	{attribute 'TcIecLibraryType'}
	{attribute 'external_name' := 'F_VN_FindContours_GUID_BC617802_F305_490B_4DCA_5F9C28F7E587'}
	(* Search for object contours in a binary image. Returns only external contours. *)
	FUNCTION F_VN_FindContours : HRESULT
	VAR_INPUT
		ipSrcImage	:	ITcVnImage;	(* Source image (modified by the function) *)
		ipContours	:	REFERENCE TO ITcVnContainer;	(* Returns a container which is filled with the found contours (ContainerType_Vector_Vector_TcVnPoint2_DINT; The elements of this container are single contours. Non-zero interface pointers are reused.) *)
		hrPrev	:	HRESULT;	(* HRESULT indicating the result of previous operations (If SUCCEEDED(hrPrev) equals false, no operation is executed.) *)
	END_VAR

END_FUNCTION

// Functions/Image Analysis/Object Detection/F_VN_FindContoursExp

	{attribute 'TcIecLibraryType'}
	{attribute 'external_name' := 'F_VN_FindContoursExp_GUID_CC63BB9E_985F_4B1D_69D1_A104A588DDE9'}
	(* Search for object contours in a binary image. (expert function) *)
	FUNCTION F_VN_FindContoursExp : HRESULT
	VAR_INPUT
		ipSrcImage	:	ITcVnImage;	(* Source image (modified by the function) *)
		ipContours	:	REFERENCE TO ITcVnContainer;	(* Returns a container which is filled with the found contours (ContainerType_Vector_Vector_TcVnPoint2_DINT; The elements of this container are single contours. Non-zero interface pointers are reused.) *)
		eRetrievalMode	:	ETcVnContourRetrievalMode;	(* Specifies which contours are retrieved and how their relationship is encoded *)
		eApproximationMethod	:	ETcVnContourApproximationMethod;	(* Contour encoding *)
		aOffset	:	REFERENCE TO TcVnPoint;	(* Offset by which every contour point is shifted *)
		hrPrev	:	HRESULT;	(* HRESULT indicating the result of previous operations (If SUCCEEDED(hrPrev) equals false, no operation is executed.) *)
	END_VAR

END_FUNCTION

// Functions/Image Analysis/Object Detection/F_VN_HoughCircles

	{attribute 'TcIecLibraryType'}
	{attribute 'external_name' := 'F_VN_HoughCircles_GUID_86F03E73_E7CE_4817_5925_A59C535A1739'}
	(* Search for circles using the Hough transform. *)
	FUNCTION F_VN_HoughCircles : HRESULT
	VAR_INPUT
		ipSrcImage	:	ITcVnImage;	(* Source image (USINT, 1 channel, gray-level) *)
		ipCircles	:	REFERENCE TO ITcVnContainer;	(* Returns a container which is filled with the found circles (ContainerType_Vector_TcVnVector3_REAL; Each container element contains the x coordinate of the circle center [0], the y coordinate of the circle center [1], and the radius [2], respectively. Non-zero interface pointers are reused.) *)
		fInvAccuRatio	:	LREAL;	(* Inverted ratio of the accumulator size in relation to the source image's size (must be > 0. A value of 2 means that the size is halved in both directions.) *)
		fMinDist	:	LREAL;	(* Smallest allowed distance of two circles (must be > 0) *)
		hrPrev	:	HRESULT;	(* HRESULT indicating the result of previous operations (If SUCCEEDED(hrPrev) equals false, no operation is executed.) *)
	END_VAR

END_FUNCTION

// Functions/Image Analysis/Object Detection/F_VN_HoughCirclesExp

	{attribute 'TcIecLibraryType'}
	{attribute 'external_name' := 'F_VN_HoughCirclesExp_GUID_B1DC5CB1_08D8_43F5_4695_748B5DA9490C'}
	(* Search for circles using the Hough transform. (expert function) *)
	FUNCTION F_VN_HoughCirclesExp : HRESULT
	VAR_INPUT
		ipSrcImage	:	ITcVnImage;	(* Source image (USINT, 1 channel, gray-level) *)
		ipCircles	:	REFERENCE TO ITcVnContainer;	(* Returns a container which is filled with the found circles (ContainerType_Vector_TcVnVector3_REAL; Each container element contains the x coordinate of the circle center [0], the y coordinate of the circle center [1], and the radius [2], respectively. Non-zero interface pointers are reused.) *)
		fInvAccuRatio	:	LREAL;	(* Inverted ratio of the accumulator size in relation to the source image's size (must be > 0. A value of 2 means that the size is halved in both directions.) *)
		fMinDist	:	LREAL;	(* Smallest allowed distance of two circles (must be > 0) *)
		eHoughMethod	:	ETcVnHoughMethod;	(* Hough method to use (currently only valid value: GRADIENT) *)
		fParam1	:	LREAL;	(* First method specific parameter (GRADIENT: upper threshold for canny edge detection, which must be > 0) *)
		fParam2	:	LREAL;	(* Second method specific parameter (GRADIENT: accumulator threshold for detecting circle centers, which must be > 0) *)
		nMinRadius	:	UDINT;	(* Minimum circle radius allowed *)
		nMaxRadius	:	UDINT;	(* Maximum circle radius allowed (if 0, the value is internally set to max(image rows, image columns)) *)
		hrPrev	:	HRESULT;	(* HRESULT indicating the result of previous operations (If SUCCEEDED(hrPrev) equals false, no operation is executed.) *)
	END_VAR

END_FUNCTION

// Functions/Image Analysis/Object Detection/F_VN_HoughLines

	{attribute 'TcIecLibraryType'}
	{attribute 'external_name' := 'F_VN_HoughLines_GUID_3641D244_03BD_44CB_43E4_F0ABC9273C89'}
	(* Search for lines using the standard Hough transform. *)
	FUNCTION F_VN_HoughLines : HRESULT
	VAR_INPUT
		ipSrcImage	:	ITcVnImage;	(* Source image (USINT, 1 channel, binary, may be modified by the function) *)
		ipLines	:	REFERENCE TO ITcVnContainer;	(* Returns a container which is filled with the found lines (ContainerType_Vector_TcVnVector2_REAL; Each container element contains the distance from the origin [0] in pixels and the rotation angle [1] in radians, respectively. Non-zero interface pointers are reused.) *)
		fDistRes	:	LREAL;	(* Distance resolution of the accumulator (in pixels, must be > 0) *)
		fAngleRes	:	LREAL;	(* Angle resolution of the accumulator (in radians, must be > 0) *)
		nAccuThreshold	:	UDINT;	(* Accumulator threshold *)
		hrPrev	:	HRESULT;	(* HRESULT indicating the result of previous operations (If SUCCEEDED(hrPrev) equals false, no operation is executed.) *)
	END_VAR

END_FUNCTION

// Functions/Image Analysis/Object Detection/F_VN_HoughLinesExp

	{attribute 'TcIecLibraryType'}
	{attribute 'external_name' := 'F_VN_HoughLinesExp_GUID_1C9FFE0A_9145_4559_5E8F_3269BB3716B9'}
	(* Search for lines using the standard Hough transform. (expert function) *)
	FUNCTION F_VN_HoughLinesExp : HRESULT
	VAR_INPUT
		ipSrcImage	:	ITcVnImage;	(* Source image (USINT, 1 channel, binary, may be modified by the function) *)
		ipLines	:	REFERENCE TO ITcVnContainer;	(* Returns a container which is filled with the found lines (ContainerType_Vector_TcVnVector2_REAL; Each container element contains the distance from the origin [0] in pixels and the rotation angle [1] in radians, respectively. Non-zero interface pointers are reused.) *)
		fDistRes	:	LREAL;	(* Distance resolution of the accumulator (in pixels, must be > 0) *)
		fAngleRes	:	LREAL;	(* Angle resolution of the accumulator (in radians, must be > 0) *)
		nAccuThreshold	:	UDINT;	(* Accumulator threshold *)
		fDistResDiv	:	LREAL;	(* Divisor of the distance resolution for the multi-scale Hough transform (>= 0, must be > 0 if fAngleResDiv is > 0) *)
		fAngleResDiv	:	LREAL;	(* Divisor of the angle resolution for the multi-scale Hough transform (>= 0, must be > 0 if fDistResDiv is > 0) *)
		hrPrev	:	HRESULT;	(* HRESULT indicating the result of previous operations (If SUCCEEDED(hrPrev) equals false, no operation is executed.) *)
	END_VAR

END_FUNCTION

// Functions/Image Analysis/Object Detection/F_VN_MatchImageHuMoments

	{attribute 'TcIecLibraryType'}
	{attribute 'external_name' := 'F_VN_MatchImageHuMoments_GUID_D174E499_AD66_4F1F_5089_AD3F3CD47605'}
	(* Compare two images using the Hu moment invariants. *)
	FUNCTION F_VN_MatchImageHuMoments : HRESULT
	VAR_INPUT
		ipImage1	:	ITcVnImage;	(* First image (1 channel) *)
		ipImage2	:	ITcVnImage;	(* Second image (1 channel) *)
		eComparisonMethod	:	ETcVnContoursMatchComparisonMethod;	(* Method used for comparing the Hu moment invariants of the images *)
		fDissimilarity	:	REFERENCE TO LREAL;	(* Returns the dissimilarity of the image Hu moment invariants depending on the chosen comparison method *)
		hrPrev	:	HRESULT;	(* HRESULT indicating the result of previous operations (If SUCCEEDED(hrPrev) equals false, no operation is executed.) *)
	END_VAR

END_FUNCTION

// Functions/Image Analysis/Object Detection/F_VN_MatchTemplate

	{attribute 'TcIecLibraryType'}
	{attribute 'external_name' := 'F_VN_MatchTemplate_GUID_741B3C57_0C32_4A22_515B_0F16608AEB4A'}
	(* Match a template image with every location in the source image (using the TCVN_TMM_CCORR_NORMED method) and save the comparison results. *)
	FUNCTION F_VN_MatchTemplate : HRESULT
	VAR_INPUT
		ipSrcImage	:	ITcVnImage;	(* Source image (USINT or REAL, 1 or 3 channels) *)
		ipTemplateImage	:	ITcVnImage;	(* Template image (same type as ipSrcImage, smaller width and height) *)
		ipResultImage	:	REFERENCE TO ITcVnImage;	(* Returns the result image (REAL, normalized to [0..1], 1 channel, dimensions: (ipSrcImage.width - ipTemplateImage.width + 1) x (ipSrcImage.height - ipTemplateImage.height + 1). The best match is the global maximum. The position in ipResultImage is the top-left corner of ipTemplateImage position in ipSrcImage) *)
		hrPrev	:	HRESULT;	(* HRESULT indicating the result of previous operations (If SUCCEEDED(hrPrev) equals false, no operation is executed.) *)
	END_VAR

END_FUNCTION

// Functions/Image Analysis/Object Detection/F_VN_MatchTemplateExp

	{attribute 'TcIecLibraryType'}
	{attribute 'external_name' := 'F_VN_MatchTemplateExp_GUID_82700BC1_22E7_489F_6AAC_8EFF22E27EF5'}
	(* Match a template image with every location in the source image and save the comparison results. (expert function) *)
	FUNCTION F_VN_MatchTemplateExp : HRESULT
	VAR_INPUT
		ipSrcImage	:	ITcVnImage;	(* Source image (USINT or REAL, 1 or 3 channels) *)
		ipTemplateImage	:	ITcVnImage;	(* Template image (same type as ipSrcImage, smaller width and height) *)
		ipResultImage	:	REFERENCE TO ITcVnImage;	(* Returns the result image (REAL, 1 channel, dimensions: (ipSrcImage.width - ipTemplateImage.width + 1) x (ipSrcImage.height - ipTemplateImage.height + 1). The best match is the global minimum (SQDIFF(_NORMED)) or maximum (CCORR(_NORMED), CCOEFF(_NORMED)). The position in ipResultImage is the top-left corner of ipTemplateImage position in ipSrcImage) *)
		eMatchMethod	:	ETcVnTemplateMatchMethod;	(* Specifies the template match method *)
		ipTemplateMask	:	ITcVnImage;	(* Optional mask for ipTemplateImage (only supported for SQDIFF and CCORR_NORMED, same type and size as ipTemplateImage) *)
		hrPrev	:	HRESULT;	(* HRESULT indicating the result of previous operations (If SUCCEEDED(hrPrev) equals false, no operation is executed.) *)
	END_VAR

END_FUNCTION

// Functions/Image Analysis/Object Detection/F_VN_MatchTemplateAndEvaluate

	{attribute 'TcIecLibraryType'}
	{attribute 'external_name' := 'F_VN_MatchTemplateAndEvaluate_GUID_6066B156_0035_483D_500E_8B9A3AFE6EDA'}
	(* Match a template image with every location in the source image (using the TCVN_TMM_CCORR_NORMED method) and evaluate the comparison results. Returns a sorted list of possible matches (best match first). *)
	FUNCTION F_VN_MatchTemplateAndEvaluate : HRESULT
	VAR_INPUT
		ipSrcImage	:	ITcVnImage;	(* Source image (USINT or REAL, 1 or 3 channels) *)
		ipTemplateImage	:	ITcVnImage;	(* Template image (same type as ipSrcImage, smaller width and height) *)
		ipMatches	:	REFERENCE TO ITcVnContainer;	(* Returns the matching positions (ContainerType_Vector_TcVnPoint2_DINT, where each element represents the top-left corner of ipTemplateImage) in ipSrcImage, sorted by relevance (best match first) *)
		fMatchThreshold	:	REAL;	(* Threshold to separate relevant from irrelevant matches (0..1, 1.0  would be a perfect match. To find a suitable value, you could evaluate some sample result images of F_VN_MatchTemplate.) *)
		hrPrev	:	HRESULT;	(* HRESULT indicating the result of previous operations (If SUCCEEDED(hrPrev) equals false, no operation is executed.) *)
	END_VAR

END_FUNCTION

// Functions/Image Analysis/Object Detection/F_VN_MatchTemplateAndEvaluateExp

	{attribute 'TcIecLibraryType'}
	{attribute 'external_name' := 'F_VN_MatchTemplateAndEvaluateExp_GUID_E68FDE05_AB07_4A67_68C5_1058AA91C26B'}
	(* Match a template image with every location in the source image and evaluate the comparison results. Returns a sorted list of possible matches (best match first). (expert function) *)
	FUNCTION F_VN_MatchTemplateAndEvaluateExp : HRESULT
	VAR_INPUT
		ipSrcImage	:	ITcVnImage;	(* Source image (USINT or REAL, 1 or 3 channels) *)
		ipTemplateImage	:	ITcVnImage;	(* Template image (same type as ipSrcImage, smaller width and height) *)
		ipMatches	:	REFERENCE TO ITcVnContainer;	(* Returns the matching positions (ContainerType_Vector_TcVnPoint2_DINT, where each element represents the top-left corner of ipTemplateImage) in ipSrcImage, sorted by relevance (best match first) *)
		fMatchThreshold	:	REAL;	(* Threshold to separate relevant from irrelevant matches (0..1 for NORMED methods, otherwise dependent on template size and content. To find a suitable value, you could evaluate some sample result images of F_VN_MatchTemplateExp.) *)
		eMatchMethod	:	ETcVnTemplateMatchMethod;	(* Specifies the template match method *)
		ipTemplateMask	:	ITcVnImage;	(* Optional mask for ipTemplateImage (only supported for SQDIFF and CCORR_NORMED, same type and size as ipTemplateImage) *)
		fScaleFactor	:	REAL;	(* Factor (0..1] to reduce source and template image width and height for better performance (but less accuracy!) *)
		eInterpolationType	:	ETcVnInterpolationType;	(* Image resize interpolation type (only used if fScaleFactor != 1, TCVN_IT_BILINEAR recommended for most cases) *)
		hrPrev	:	HRESULT;	(* HRESULT indicating the result of previous operations (If SUCCEEDED(hrPrev) equals false, no operation is executed.) *)
	END_VAR

END_FUNCTION

// Functions/Basic Container Operations/F_VN_AppendToContainer/F_VN_AppendToContainer_ITcVnContainer

	{attribute 'TcIecLibraryType'}
	{attribute 'external_name' := 'F_VN_AppendToContainer_ITcVnContainer_GUID_BC895C73_8F6D_4E37_41EA_51A0EC176B08'}
	(* Append a single element to a container or concatenate containers (if ipElement has the same typeId as ipContainer). *)
	FUNCTION F_VN_AppendToContainer_ITcVnContainer : HRESULT
	VAR_INPUT
		ipElement	:	ITcVnContainer;	(* Single element to append to ipContainer or container with several elements to be concatenated *)
		ipContainer	:	ITcVnContainer;	(* Container to which the element(s) will be appended *)
		hrPrev	:	HRESULT;	(* HRESULT indicating the result of previous operations (If SUCCEEDED(hrPrev) equals false, no operation is executed.) *)
	END_VAR

END_FUNCTION

// Functions/Basic Container Operations/F_VN_AppendToContainer/F_VN_AppendToContainer_ITcVnForwardIterator

	{attribute 'TcIecLibraryType'}
	{attribute 'external_name' := 'F_VN_AppendToContainer_ITcVnForwardIterator_GUID_DC06B651_1309_4C97_69B4_24FDEC04B60D'}
	(* Append a single element (represented by an iterator)to a container. *)
	FUNCTION F_VN_AppendToContainer_ITcVnForwardIterator : HRESULT
	VAR_INPUT
		ipElement	:	ITcVnForwardIterator;	(* Single element to append to ipContainer *)
		ipContainer	:	ITcVnContainer;	(* Container to which the element(s) will be appended *)
		hrPrev	:	HRESULT;	(* HRESULT indicating the result of previous operations (If SUCCEEDED(hrPrev) equals false, no operation is executed.) *)
	END_VAR

END_FUNCTION

// Functions/Basic Container Operations/F_VN_AppendToContainer/F_VN_AppendToContainer_LREAL

	{attribute 'TcIecLibraryType'}
	{attribute 'external_name' := 'F_VN_AppendToContainer_LREAL_GUID_86D67860_56E2_4042_45E7_5CDEAC85E231'}
	(* Append a single element of type LREAL to a container. *)
	FUNCTION F_VN_AppendToContainer_LREAL : HRESULT
	VAR_INPUT
		fElement	:	LREAL;	(* Single element to append to ipContainer *)
		ipContainer	:	ITcVnContainer;	(* Container to which the element will be appended *)
		hrPrev	:	HRESULT;	(* HRESULT indicating the result of previous operations (If SUCCEEDED(hrPrev) equals false, no operation is executed.) *)
	END_VAR

END_FUNCTION

// Functions/Basic Container Operations/F_VN_AppendToContainer/F_VN_AppendToContainer_REAL

	{attribute 'TcIecLibraryType'}
	{attribute 'external_name' := 'F_VN_AppendToContainer_REAL_GUID_9FD3A03F_1D25_46B6_5C63_994ECFCB7D9B'}
	(* Append a single element of type REAL to a container. *)
	FUNCTION F_VN_AppendToContainer_REAL : HRESULT
	VAR_INPUT
		fElement	:	REAL;	(* Single element to append to ipContainer *)
		ipContainer	:	ITcVnContainer;	(* Container to which the element will be appended *)
		hrPrev	:	HRESULT;	(* HRESULT indicating the result of previous operations (If SUCCEEDED(hrPrev) equals false, no operation is executed.) *)
	END_VAR

END_FUNCTION

// Functions/Basic Container Operations/F_VN_AppendToContainer/F_VN_AppendToContainer_SINT

	{attribute 'TcIecLibraryType'}
	{attribute 'external_name' := 'F_VN_AppendToContainer_SINT_GUID_19F63135_AFAE_4A1C_5884_F4977170C8E9'}
	(* Append a single element of type SINT to a container. *)
	FUNCTION F_VN_AppendToContainer_SINT : HRESULT
	VAR_INPUT
		nElement	:	SINT;	(* Single element to append to ipContainer *)
		ipContainer	:	ITcVnContainer;	(* Container to which the element will be appended *)
		hrPrev	:	HRESULT;	(* HRESULT indicating the result of previous operations (If SUCCEEDED(hrPrev) equals false, no operation is executed.) *)
	END_VAR

END_FUNCTION

// Functions/Basic Container Operations/F_VN_AppendToContainer/F_VN_AppendToContainer_TcVnDMatch

	{attribute 'TcIecLibraryType'}
	{attribute 'external_name' := 'F_VN_AppendToContainer_TcVnDMatch_GUID_03F0054A_EBF9_4D93_55D7_76FF2D559017'}
	(* Append a single element of type TcVnDMatch to a container. *)
	FUNCTION F_VN_AppendToContainer_TcVnDMatch : HRESULT
	VAR_INPUT
		stElement	:	REFERENCE TO TcVnDMatch;	(* Single element to append to ipContainer *)
		ipContainer	:	ITcVnContainer;	(* Container to which the element will be appended *)
		hrPrev	:	HRESULT;	(* HRESULT indicating the result of previous operations (If SUCCEEDED(hrPrev) equals false, no operation is executed.) *)
	END_VAR

END_FUNCTION

// Functions/Basic Container Operations/F_VN_AppendToContainer/F_VN_AppendToContainer_TcVnKeyPoint

	{attribute 'TcIecLibraryType'}
	{attribute 'external_name' := 'F_VN_AppendToContainer_TcVnKeyPoint_GUID_EA6806AE_C5C4_48B0_4044_CCB94CE824FB'}
	(* Append a single element of type TcVnKeyPoint to a container. *)
	FUNCTION F_VN_AppendToContainer_TcVnKeyPoint : HRESULT
	VAR_INPUT
		stElement	:	REFERENCE TO TcVnKeyPoint;	(* Single element to append to ipContainer *)
		ipContainer	:	ITcVnContainer;	(* Container to which the element will be appended *)
		hrPrev	:	HRESULT;	(* HRESULT indicating the result of previous operations (If SUCCEEDED(hrPrev) equals false, no operation is executed.) *)
	END_VAR

END_FUNCTION

// Functions/Basic Container Operations/F_VN_AppendToContainer/F_VN_AppendToContainer_TcVnPoint2_DINT

	{attribute 'TcIecLibraryType'}
	{attribute 'external_name' := 'F_VN_AppendToContainer_TcVnPoint2_DINT_GUID_D542BC36_5107_4126_728B_39B063CEEFF1'}
	(* Append a single element of type TcVnPoint2_DINT to a container. *)
	FUNCTION F_VN_AppendToContainer_TcVnPoint2_DINT : HRESULT
	VAR_INPUT
		aElement	:	REFERENCE TO TcVnPoint2_DINT;	(* Single element to append to ipContainer *)
		ipContainer	:	ITcVnContainer;	(* Container to which the element will be appended *)
		hrPrev	:	HRESULT;	(* HRESULT indicating the result of previous operations (If SUCCEEDED(hrPrev) equals false, no operation is executed.) *)
	END_VAR

END_FUNCTION

// Functions/Basic Container Operations/F_VN_AppendToContainer/F_VN_AppendToContainer_TcVnPoint2_LREAL

	{attribute 'TcIecLibraryType'}
	{attribute 'external_name' := 'F_VN_AppendToContainer_TcVnPoint2_LREAL_GUID_21805E10_2AA9_48F0_6A10_EF0B16BAC43A'}
	(* Append a single element of type TcVnPoint2_LREAL to a container. *)
	FUNCTION F_VN_AppendToContainer_TcVnPoint2_LREAL : HRESULT
	VAR_INPUT
		aElement	:	REFERENCE TO TcVnPoint2_LREAL;	(* Single element to append to ipContainer *)
		ipContainer	:	ITcVnContainer;	(* Container to which the element will be appended *)
		hrPrev	:	HRESULT;	(* HRESULT indicating the result of previous operations (If SUCCEEDED(hrPrev) equals false, no operation is executed.) *)
	END_VAR

END_FUNCTION

// Functions/Basic Container Operations/F_VN_AppendToContainer/F_VN_AppendToContainer_TcVnPoint2_REAL

	{attribute 'TcIecLibraryType'}
	{attribute 'external_name' := 'F_VN_AppendToContainer_TcVnPoint2_REAL_GUID_98543EB2_5630_4CBE_4166_49DF3A89C470'}
	(* Append a single element of type TcVnPoint2_REAL to a container. *)
	FUNCTION F_VN_AppendToContainer_TcVnPoint2_REAL : HRESULT
	VAR_INPUT
		aElement	:	REFERENCE TO TcVnPoint2_REAL;	(* Single element to append to ipContainer *)
		ipContainer	:	ITcVnContainer;	(* Container to which the element will be appended *)
		hrPrev	:	HRESULT;	(* HRESULT indicating the result of previous operations (If SUCCEEDED(hrPrev) equals false, no operation is executed.) *)
	END_VAR

END_FUNCTION

// Functions/Basic Container Operations/F_VN_AppendToContainer/F_VN_AppendToContainer_TcVnPoint3_LREAL

	{attribute 'TcIecLibraryType'}
	{attribute 'external_name' := 'F_VN_AppendToContainer_TcVnPoint3_LREAL_GUID_74F53FA8_A651_4F81_609E_407D39BA6D5E'}
	(* Append a single element of type TcVnPoint3_LREAL to a container. *)
	FUNCTION F_VN_AppendToContainer_TcVnPoint3_LREAL : HRESULT
	VAR_INPUT
		aElement	:	REFERENCE TO TcVnPoint3_LREAL;	(* Single element to append to ipContainer *)
		ipContainer	:	ITcVnContainer;	(* Container to which the element will be appended *)
		hrPrev	:	HRESULT;	(* HRESULT indicating the result of previous operations (If SUCCEEDED(hrPrev) equals false, no operation is executed.) *)
	END_VAR

END_FUNCTION

// Functions/Basic Container Operations/F_VN_AppendToContainer/F_VN_AppendToContainer_TcVnPoint3_REAL

	{attribute 'TcIecLibraryType'}
	{attribute 'external_name' := 'F_VN_AppendToContainer_TcVnPoint3_REAL_GUID_682DAD9C_E660_483F_7C4E_073C42E7EE69'}
	(* Append a single element of type TcVnPoint3_REAL to a container. *)
	FUNCTION F_VN_AppendToContainer_TcVnPoint3_REAL : HRESULT
	VAR_INPUT
		aElement	:	REFERENCE TO TcVnPoint3_REAL;	(* Single element to append to ipContainer *)
		ipContainer	:	ITcVnContainer;	(* Container to which the element will be appended *)
		hrPrev	:	HRESULT;	(* HRESULT indicating the result of previous operations (If SUCCEEDED(hrPrev) equals false, no operation is executed.) *)
	END_VAR

END_FUNCTION

// Functions/Basic Container Operations/F_VN_AppendToContainer/F_VN_AppendToContainer_TcVnRectangle_DINT

	{attribute 'TcIecLibraryType'}
	{attribute 'external_name' := 'F_VN_AppendToContainer_TcVnRectangle_DINT_GUID_70508A72_C9A6_4A7D_6ACE_1A226A1C92CA'}
	(* Append a single element of type TcVnRectangle_DINT to a container. *)
	FUNCTION F_VN_AppendToContainer_TcVnRectangle_DINT : HRESULT
	VAR_INPUT
		stElement	:	REFERENCE TO TcVnRectangle_DINT;	(* Single element to append to ipContainer *)
		ipContainer	:	ITcVnContainer;	(* Container to which the element will be appended *)
		hrPrev	:	HRESULT;	(* HRESULT indicating the result of previous operations (If SUCCEEDED(hrPrev) equals false, no operation is executed.) *)
	END_VAR

END_FUNCTION

// Functions/Basic Container Operations/F_VN_AppendToContainer/F_VN_AppendToContainer_TcVnVector2_DINT

	{attribute 'TcIecLibraryType'}
	{attribute 'external_name' := 'F_VN_AppendToContainer_TcVnVector2_DINT_GUID_F54BDCBC_4F9C_4BFF_5F0D_9BBA1ECF64E1'}
	(* Append a single element of type TcVnVector2_DINT to a container. *)
	FUNCTION F_VN_AppendToContainer_TcVnVector2_DINT : HRESULT
	VAR_INPUT
		aElement	:	REFERENCE TO TcVnVector2_DINT;	(* Single element to append to ipContainer *)
		ipContainer	:	ITcVnContainer;	(* Container to which the element will be appended *)
		hrPrev	:	HRESULT;	(* HRESULT indicating the result of previous operations (If SUCCEEDED(hrPrev) equals false, no operation is executed.) *)
	END_VAR

END_FUNCTION

// Functions/Basic Container Operations/F_VN_AppendToContainer/F_VN_AppendToContainer_TcVnVector2_REAL

	{attribute 'TcIecLibraryType'}
	{attribute 'external_name' := 'F_VN_AppendToContainer_TcVnVector2_REAL_GUID_7E5185E2_3C3A_4A6D_410E_85FFF2DDA7ED'}
	(* Append a single element of type TcVnVector2_REAL to a container. *)
	FUNCTION F_VN_AppendToContainer_TcVnVector2_REAL : HRESULT
	VAR_INPUT
		aElement	:	REFERENCE TO TcVnVector2_REAL;	(* Single element to append to ipContainer *)
		ipContainer	:	ITcVnContainer;	(* Container to which the element will be appended *)
		hrPrev	:	HRESULT;	(* HRESULT indicating the result of previous operations (If SUCCEEDED(hrPrev) equals false, no operation is executed.) *)
	END_VAR

END_FUNCTION

// Functions/Basic Container Operations/F_VN_AppendToContainer/F_VN_AppendToContainer_TcVnVector3_REAL

	{attribute 'TcIecLibraryType'}
	{attribute 'external_name' := 'F_VN_AppendToContainer_TcVnVector3_REAL_GUID_66346CA2_B066_4C43_7176_A73748BB3D6B'}
	(* Append a single element of type TcVnVector3_REAL to a container. *)
	FUNCTION F_VN_AppendToContainer_TcVnVector3_REAL : HRESULT
	VAR_INPUT
		aElement	:	REFERENCE TO TcVnVector3_REAL;	(* Single element to append to ipContainer *)
		ipContainer	:	ITcVnContainer;	(* Container to which the element will be appended *)
		hrPrev	:	HRESULT;	(* HRESULT indicating the result of previous operations (If SUCCEEDED(hrPrev) equals false, no operation is executed.) *)
	END_VAR

END_FUNCTION

// Functions/Basic Container Operations/F_VN_AppendToContainer/F_VN_AppendToContainer_TcVnVector4_DINT

	{attribute 'TcIecLibraryType'}
	{attribute 'external_name' := 'F_VN_AppendToContainer_TcVnVector4_DINT_GUID_3F4B7132_C6F5_42F5_5AA6_2B5EFE9FD284'}
	(* Append a single element of type TcVnVector4_DINT to a container. *)
	FUNCTION F_VN_AppendToContainer_TcVnVector4_DINT : HRESULT
	VAR_INPUT
		aElement	:	REFERENCE TO TcVnVector4_DINT;	(* Single element to append to ipContainer *)
		ipContainer	:	ITcVnContainer;	(* Container to which the element will be appended *)
		hrPrev	:	HRESULT;	(* HRESULT indicating the result of previous operations (If SUCCEEDED(hrPrev) equals false, no operation is executed.) *)
	END_VAR

END_FUNCTION

// Functions/Basic Container Operations/F_VN_AppendToContainer/F_VN_AppendToContainer_UDINT

	{attribute 'TcIecLibraryType'}
	{attribute 'external_name' := 'F_VN_AppendToContainer_UDINT_GUID_B3048746_2673_4E23_668E_25707083473A'}
	(* Append a single element of type UDINT to a container. *)
	FUNCTION F_VN_AppendToContainer_UDINT : HRESULT
	VAR_INPUT
		nElement	:	UDINT;	(* Single element to append to ipContainer *)
		ipContainer	:	ITcVnContainer;	(* Container to which the element will be appended *)
		hrPrev	:	HRESULT;	(* HRESULT indicating the result of previous operations (If SUCCEEDED(hrPrev) equals false, no operation is executed.) *)
	END_VAR

END_FUNCTION

// Functions/Basic Container Operations/F_VN_AppendToContainer/F_VN_AppendToContainer_ULINT

	{attribute 'TcIecLibraryType'}
	{attribute 'external_name' := 'F_VN_AppendToContainer_ULINT_GUID_8552DB7D_4165_4A8D_5303_28A530C24467'}
	(* Append a single element of type ULINT to a container. *)
	FUNCTION F_VN_AppendToContainer_ULINT : HRESULT
	VAR_INPUT
		nElement	:	ULINT;	(* Single element to append to ipContainer *)
		ipContainer	:	ITcVnContainer;	(* Container to which the element will be appended *)
		hrPrev	:	HRESULT;	(* HRESULT indicating the result of previous operations (If SUCCEEDED(hrPrev) equals false, no operation is executed.) *)
	END_VAR

END_FUNCTION

// Functions/Basic Container Operations/F_VN_FillContainer/F_VN_FillContainer_LREAL

	{attribute 'TcIecLibraryType'}
	{attribute 'external_name' := 'F_VN_FillContainer_LREAL_GUID_BA4B68D0_82F5_477F_4679_4180419A472B'}
	(* Fill the container with the specified value. Only possible for containers with basic elements. *)
	FUNCTION F_VN_FillContainer_LREAL : HRESULT
	VAR_INPUT
		ipContainer	:	ITcVnContainer;	(* Container with basic elements *)
		fValue	:	LREAL;	(* Value to set the container elements *)
		hrPrev	:	HRESULT;	(* HRESULT indicating the result of previous operations (If SUCCEEDED(hrPrev) equals false, no operation is executed.) *)
	END_VAR

END_FUNCTION

// Functions/Basic Container Operations/F_VN_FillContainer/F_VN_FillContainer_REAL

	{attribute 'TcIecLibraryType'}
	{attribute 'external_name' := 'F_VN_FillContainer_REAL_GUID_E7414682_9BD2_4DA6_78C1_D2E1E2508E11'}
	(* Fill the container with the specified value. Only possible for containers with basic elements. *)
	FUNCTION F_VN_FillContainer_REAL : HRESULT
	VAR_INPUT
		ipContainer	:	ITcVnContainer;	(* Container with basic elements *)
		fValue	:	REAL;	(* Value to set the container elements *)
		hrPrev	:	HRESULT;	(* HRESULT indicating the result of previous operations (If SUCCEEDED(hrPrev) equals false, no operation is executed.) *)
	END_VAR

END_FUNCTION

// Functions/Basic Container Operations/F_VN_FillContainer/F_VN_FillContainer_SINT

	{attribute 'TcIecLibraryType'}
	{attribute 'external_name' := 'F_VN_FillContainer_SINT_GUID_C07D0195_EC31_4F82_4A4E_E15E801A7424'}
	(* Fill the container with the specified value. Only possible for containers with basic elements. *)
	FUNCTION F_VN_FillContainer_SINT : HRESULT
	VAR_INPUT
		ipContainer	:	ITcVnContainer;	(* Container with basic elements *)
		nValue	:	SINT;	(* Value to set the container elements *)
		hrPrev	:	HRESULT;	(* HRESULT indicating the result of previous operations (If SUCCEEDED(hrPrev) equals false, no operation is executed.) *)
	END_VAR

END_FUNCTION

// Functions/Basic Container Operations/F_VN_FillContainer/F_VN_FillContainer_TcVnDMatch

	{attribute 'TcIecLibraryType'}
	{attribute 'external_name' := 'F_VN_FillContainer_TcVnDMatch_GUID_ADBDB5A7_9332_4BD4_4D6B_209FBD6606EC'}
	(* Fill the container with the specified value. Only possible for containers with basic elements. *)
	FUNCTION F_VN_FillContainer_TcVnDMatch : HRESULT
	VAR_INPUT
		ipContainer	:	ITcVnContainer;	(* Container with basic elements *)
		stValue	:	REFERENCE TO TcVnDMatch;	(* Value to set the container elements *)
		hrPrev	:	HRESULT;	(* HRESULT indicating the result of previous operations (If SUCCEEDED(hrPrev) equals false, no operation is executed.) *)
	END_VAR

END_FUNCTION

// Functions/Basic Container Operations/F_VN_FillContainer/F_VN_FillContainer_TcVnKeyPoint

	{attribute 'TcIecLibraryType'}
	{attribute 'external_name' := 'F_VN_FillContainer_TcVnKeyPoint_GUID_270DFBB3_EDBD_4E87_448A_4B20AEF05EFB'}
	(* Fill the container with the specified value. Only possible for containers with basic elements. *)
	FUNCTION F_VN_FillContainer_TcVnKeyPoint : HRESULT
	VAR_INPUT
		ipContainer	:	ITcVnContainer;	(* Container with basic elements *)
		stValue	:	REFERENCE TO TcVnKeyPoint;	(* Value to set the container elements *)
		hrPrev	:	HRESULT;	(* HRESULT indicating the result of previous operations (If SUCCEEDED(hrPrev) equals false, no operation is executed.) *)
	END_VAR

END_FUNCTION

// Functions/Basic Container Operations/F_VN_FillContainer/F_VN_FillContainer_TcVnPoint2_DINT

	{attribute 'TcIecLibraryType'}
	{attribute 'external_name' := 'F_VN_FillContainer_TcVnPoint2_DINT_GUID_3D9234EF_11A6_46F7_4B47_E9026B7E311A'}
	(* Fill the container with the specified value. Only possible for containers with basic elements. *)
	FUNCTION F_VN_FillContainer_TcVnPoint2_DINT : HRESULT
	VAR_INPUT
		ipContainer	:	ITcVnContainer;	(* Container with basic elements *)
		aValue	:	REFERENCE TO TcVnPoint2_DINT;	(* Value to set the container elements *)
		hrPrev	:	HRESULT;	(* HRESULT indicating the result of previous operations (If SUCCEEDED(hrPrev) equals false, no operation is executed.) *)
	END_VAR

END_FUNCTION

// Functions/Basic Container Operations/F_VN_FillContainer/F_VN_FillContainer_TcVnPoint2_LREAL

	{attribute 'TcIecLibraryType'}
	{attribute 'external_name' := 'F_VN_FillContainer_TcVnPoint2_LREAL_GUID_9D4FC182_CFB2_409B_62F1_32576C3B99D8'}
	(* Fill the container with the specified value. Only possible for containers with basic elements. *)
	FUNCTION F_VN_FillContainer_TcVnPoint2_LREAL : HRESULT
	VAR_INPUT
		ipContainer	:	ITcVnContainer;	(* Container with basic elements *)
		aValue	:	REFERENCE TO TcVnPoint2_LREAL;	(* Value to set the container elements *)
		hrPrev	:	HRESULT;	(* HRESULT indicating the result of previous operations (If SUCCEEDED(hrPrev) equals false, no operation is executed.) *)
	END_VAR

END_FUNCTION

// Functions/Basic Container Operations/F_VN_FillContainer/F_VN_FillContainer_TcVnPoint2_REAL

	{attribute 'TcIecLibraryType'}
	{attribute 'external_name' := 'F_VN_FillContainer_TcVnPoint2_REAL_GUID_32FE7D28_1185_4A59_4D15_59D423477EEB'}
	(* Fill the container with the specified value. Only possible for containers with basic elements. *)
	FUNCTION F_VN_FillContainer_TcVnPoint2_REAL : HRESULT
	VAR_INPUT
		ipContainer	:	ITcVnContainer;	(* Container with basic elements *)
		aValue	:	REFERENCE TO TcVnPoint2_REAL;	(* Value to set the container elements *)
		hrPrev	:	HRESULT;	(* HRESULT indicating the result of previous operations (If SUCCEEDED(hrPrev) equals false, no operation is executed.) *)
	END_VAR

END_FUNCTION

// Functions/Basic Container Operations/F_VN_FillContainer/F_VN_FillContainer_TcVnPoint3_LREAL

	{attribute 'TcIecLibraryType'}
	{attribute 'external_name' := 'F_VN_FillContainer_TcVnPoint3_LREAL_GUID_C9BE38BF_16C0_4E2C_7BC6_7CB586A2B95D'}
	(* Fill the container with the specified value. Only possible for containers with basic elements. *)
	FUNCTION F_VN_FillContainer_TcVnPoint3_LREAL : HRESULT
	VAR_INPUT
		ipContainer	:	ITcVnContainer;	(* Container with basic elements *)
		aValue	:	REFERENCE TO TcVnPoint3_LREAL;	(* Value to set the container elements *)
		hrPrev	:	HRESULT;	(* HRESULT indicating the result of previous operations (If SUCCEEDED(hrPrev) equals false, no operation is executed.) *)
	END_VAR

END_FUNCTION

// Functions/Basic Container Operations/F_VN_FillContainer/F_VN_FillContainer_TcVnPoint3_REAL

	{attribute 'TcIecLibraryType'}
	{attribute 'external_name' := 'F_VN_FillContainer_TcVnPoint3_REAL_GUID_2837DBCC_797F_4F96_4168_659321D1341E'}
	(* Fill the container with the specified value. Only possible for containers with basic elements. *)
	FUNCTION F_VN_FillContainer_TcVnPoint3_REAL : HRESULT
	VAR_INPUT
		ipContainer	:	ITcVnContainer;	(* Container with basic elements *)
		aValue	:	REFERENCE TO TcVnPoint3_REAL;	(* Value to set the container elements *)
		hrPrev	:	HRESULT;	(* HRESULT indicating the result of previous operations (If SUCCEEDED(hrPrev) equals false, no operation is executed.) *)
	END_VAR

END_FUNCTION

// Functions/Basic Container Operations/F_VN_FillContainer/F_VN_FillContainer_TcVnRectangle_DINT

	{attribute 'TcIecLibraryType'}
	{attribute 'external_name' := 'F_VN_FillContainer_TcVnRectangle_DINT_GUID_58FEF820_3008_4367_6577_42BCF32C72F8'}
	(* Fill the container with the specified value. Only possible for containers with basic elements. *)
	FUNCTION F_VN_FillContainer_TcVnRectangle_DINT : HRESULT
	VAR_INPUT
		ipContainer	:	ITcVnContainer;	(* Container with basic elements *)
		stValue	:	REFERENCE TO TcVnRectangle_DINT;	(* Value to set the container elements *)
		hrPrev	:	HRESULT;	(* HRESULT indicating the result of previous operations (If SUCCEEDED(hrPrev) equals false, no operation is executed.) *)
	END_VAR

END_FUNCTION

// Functions/Basic Container Operations/F_VN_FillContainer/F_VN_FillContainer_TcVnVector2_DINT

	{attribute 'TcIecLibraryType'}
	{attribute 'external_name' := 'F_VN_FillContainer_TcVnVector2_DINT_GUID_626AF193_9CD3_491D_624F_26F1E66DEE43'}
	(* Fill the container with the specified value. Only possible for containers with basic elements. *)
	FUNCTION F_VN_FillContainer_TcVnVector2_DINT : HRESULT
	VAR_INPUT
		ipContainer	:	ITcVnContainer;	(* Container with basic elements *)
		aValue	:	REFERENCE TO TcVnVector2_DINT;	(* Value to set the container elements *)
		hrPrev	:	HRESULT;	(* HRESULT indicating the result of previous operations (If SUCCEEDED(hrPrev) equals false, no operation is executed.) *)
	END_VAR

END_FUNCTION

// Functions/Basic Container Operations/F_VN_FillContainer/F_VN_FillContainer_TcVnVector2_REAL

	{attribute 'TcIecLibraryType'}
	{attribute 'external_name' := 'F_VN_FillContainer_TcVnVector2_REAL_GUID_F5AB9681_829D_47A2_5145_D9A9E901E427'}
	(* Fill the container with the specified value. Only possible for containers with basic elements. *)
	FUNCTION F_VN_FillContainer_TcVnVector2_REAL : HRESULT
	VAR_INPUT
		ipContainer	:	ITcVnContainer;	(* Container with basic elements *)
		aValue	:	REFERENCE TO TcVnVector2_REAL;	(* Value to set the container elements *)
		hrPrev	:	HRESULT;	(* HRESULT indicating the result of previous operations (If SUCCEEDED(hrPrev) equals false, no operation is executed.) *)
	END_VAR

END_FUNCTION

// Functions/Basic Container Operations/F_VN_FillContainer/F_VN_FillContainer_TcVnVector3_REAL

	{attribute 'TcIecLibraryType'}
	{attribute 'external_name' := 'F_VN_FillContainer_TcVnVector3_REAL_GUID_AC4DD3D5_F641_4E54_6FBC_747824F29F91'}
	(* Fill the container with the specified value. Only possible for containers with basic elements. *)
	FUNCTION F_VN_FillContainer_TcVnVector3_REAL : HRESULT
	VAR_INPUT
		ipContainer	:	ITcVnContainer;	(* Container with basic elements *)
		aValue	:	REFERENCE TO TcVnVector3_REAL;	(* Value to set the container elements *)
		hrPrev	:	HRESULT;	(* HRESULT indicating the result of previous operations (If SUCCEEDED(hrPrev) equals false, no operation is executed.) *)
	END_VAR

END_FUNCTION

// Functions/Basic Container Operations/F_VN_FillContainer/F_VN_FillContainer_TcVnVector4_DINT

	{attribute 'TcIecLibraryType'}
	{attribute 'external_name' := 'F_VN_FillContainer_TcVnVector4_DINT_GUID_A36C46F6_4B94_4974_49EE_460399855F7E'}
	(* Fill the container with the specified value. Only possible for containers with basic elements. *)
	FUNCTION F_VN_FillContainer_TcVnVector4_DINT : HRESULT
	VAR_INPUT
		ipContainer	:	ITcVnContainer;	(* Container with basic elements *)
		aValue	:	REFERENCE TO TcVnVector4_DINT;	(* Value to set the container elements *)
		hrPrev	:	HRESULT;	(* HRESULT indicating the result of previous operations (If SUCCEEDED(hrPrev) equals false, no operation is executed.) *)
	END_VAR

END_FUNCTION

// Functions/Basic Container Operations/F_VN_FillContainer/F_VN_FillContainer_UDINT

	{attribute 'TcIecLibraryType'}
	{attribute 'external_name' := 'F_VN_FillContainer_UDINT_GUID_14E30BA9_473B_49EF_630E_ED6474F497BB'}
	(* Fill the container with the specified value. Only possible for containers with basic elements. *)
	FUNCTION F_VN_FillContainer_UDINT : HRESULT
	VAR_INPUT
		ipContainer	:	ITcVnContainer;	(* Container with basic elements *)
		nValue	:	UDINT;	(* Value to set the container elements *)
		hrPrev	:	HRESULT;	(* HRESULT indicating the result of previous operations (If SUCCEEDED(hrPrev) equals false, no operation is executed.) *)
	END_VAR

END_FUNCTION

// Functions/Basic Container Operations/F_VN_FillContainer/F_VN_FillContainer_ULINT

	{attribute 'TcIecLibraryType'}
	{attribute 'external_name' := 'F_VN_FillContainer_ULINT_GUID_296B9D94_9BF8_4A0E_4799_CBB907633BDB'}
	(* Fill the container with the specified value. Only possible for containers with basic elements. *)
	FUNCTION F_VN_FillContainer_ULINT : HRESULT
	VAR_INPUT
		ipContainer	:	ITcVnContainer;	(* Container with basic elements *)
		nValue	:	ULINT;	(* Value to set the container elements *)
		hrPrev	:	HRESULT;	(* HRESULT indicating the result of previous operations (If SUCCEEDED(hrPrev) equals false, no operation is executed.) *)
	END_VAR

END_FUNCTION

// Functions/Basic Container Operations/F_VN_FillContainerExp/F_VN_FillContainerExp_LREAL

	{attribute 'TcIecLibraryType'}
	{attribute 'external_name' := 'F_VN_FillContainerExp_LREAL_GUID_46711F8F_93E9_469C_40CA_BB16749B0207'}
	(* Partially fill the container with the specified value. Only possible for containers with basic elements. (expert function) *)
	FUNCTION F_VN_FillContainerExp_LREAL : HRESULT
	VAR_INPUT
		ipContainer	:	ITcVnContainer;	(* Container with basic elements *)
		fValue	:	LREAL;	(* Value to set the container elements *)
		nStartIdx	:	ULINT;	(* Start index *)
		nCount	:	ULINT;	(* Number of elements to set *)
		hrPrev	:	HRESULT;	(* HRESULT indicating the result of previous operations (If SUCCEEDED(hrPrev) equals false, no operation is executed.) *)
	END_VAR

END_FUNCTION

// Functions/Basic Container Operations/F_VN_FillContainerExp/F_VN_FillContainerExp_REAL

	{attribute 'TcIecLibraryType'}
	{attribute 'external_name' := 'F_VN_FillContainerExp_REAL_GUID_0861AC98_893D_4556_700F_2CE8CE1F7BD4'}
	(* Partially fill the container with the specified value. Only possible for containers with basic elements. (expert function) *)
	FUNCTION F_VN_FillContainerExp_REAL : HRESULT
	VAR_INPUT
		ipContainer	:	ITcVnContainer;	(* Container with basic elements *)
		fValue	:	REAL;	(* Value to set the container elements *)
		nStartIdx	:	ULINT;	(* Start index *)
		nCount	:	ULINT;	(* Number of elements to set *)
		hrPrev	:	HRESULT;	(* HRESULT indicating the result of previous operations (If SUCCEEDED(hrPrev) equals false, no operation is executed.) *)
	END_VAR

END_FUNCTION

// Functions/Basic Container Operations/F_VN_FillContainerExp/F_VN_FillContainerExp_SINT

	{attribute 'TcIecLibraryType'}
	{attribute 'external_name' := 'F_VN_FillContainerExp_SINT_GUID_D05FD693_0E6B_485A_7AFB_9BF4FFC8FFB0'}
	(* Partially fill the container with the specified value. Only possible for containers with basic elements. (expert function) *)
	FUNCTION F_VN_FillContainerExp_SINT : HRESULT
	VAR_INPUT
		ipContainer	:	ITcVnContainer;	(* Container with basic elements *)
		nValue	:	SINT;	(* Value to set the container elements *)
		nStartIdx	:	ULINT;	(* Start index *)
		nCount	:	ULINT;	(* Number of elements to set *)
		hrPrev	:	HRESULT;	(* HRESULT indicating the result of previous operations (If SUCCEEDED(hrPrev) equals false, no operation is executed.) *)
	END_VAR

END_FUNCTION

// Functions/Basic Container Operations/F_VN_FillContainerExp/F_VN_FillContainerExp_TcVnDMatch

	{attribute 'TcIecLibraryType'}
	{attribute 'external_name' := 'F_VN_FillContainerExp_TcVnDMatch_GUID_2E6AC373_8603_48DB_6DDE_414662F84002'}
	(* Partially fill the container with the specified value. Only possible for containers with basic elements. (expert function) *)
	FUNCTION F_VN_FillContainerExp_TcVnDMatch : HRESULT
	VAR_INPUT
		ipContainer	:	ITcVnContainer;	(* Container with basic elements *)
		stValue	:	REFERENCE TO TcVnDMatch;	(* Value to set the container elements *)
		nStartIdx	:	ULINT;	(* Start index *)
		nCount	:	ULINT;	(* Number of elements to set *)
		hrPrev	:	HRESULT;	(* HRESULT indicating the result of previous operations (If SUCCEEDED(hrPrev) equals false, no operation is executed.) *)
	END_VAR

END_FUNCTION

// Functions/Basic Container Operations/F_VN_FillContainerExp/F_VN_FillContainerExp_TcVnKeyPoint

	{attribute 'TcIecLibraryType'}
	{attribute 'external_name' := 'F_VN_FillContainerExp_TcVnKeyPoint_GUID_1E550ECC_9036_44EC_49BD_27256B88E7EF'}
	(* Partially fill the container with the specified value. Only possible for containers with basic elements. (expert function) *)
	FUNCTION F_VN_FillContainerExp_TcVnKeyPoint : HRESULT
	VAR_INPUT
		ipContainer	:	ITcVnContainer;	(* Container with basic elements *)
		stValue	:	REFERENCE TO TcVnKeyPoint;	(* Value to set the container elements *)
		nStartIdx	:	ULINT;	(* Start index *)
		nCount	:	ULINT;	(* Number of elements to set *)
		hrPrev	:	HRESULT;	(* HRESULT indicating the result of previous operations (If SUCCEEDED(hrPrev) equals false, no operation is executed.) *)
	END_VAR

END_FUNCTION

// Functions/Basic Container Operations/F_VN_FillContainerExp/F_VN_FillContainerExp_TcVnPoint2_DINT

	{attribute 'TcIecLibraryType'}
	{attribute 'external_name' := 'F_VN_FillContainerExp_TcVnPoint2_DINT_GUID_152069C9_A826_489E_5737_BF117E50970F'}
	(* Partially fill the container with the specified value. Only possible for containers with basic elements. (expert function) *)
	FUNCTION F_VN_FillContainerExp_TcVnPoint2_DINT : HRESULT
	VAR_INPUT
		ipContainer	:	ITcVnContainer;	(* Container with basic elements *)
		aValue	:	REFERENCE TO TcVnPoint2_DINT;	(* Value to set the container elements *)
		nStartIdx	:	ULINT;	(* Start index *)
		nCount	:	ULINT;	(* Number of elements to set *)
		hrPrev	:	HRESULT;	(* HRESULT indicating the result of previous operations (If SUCCEEDED(hrPrev) equals false, no operation is executed.) *)
	END_VAR

END_FUNCTION

// Functions/Basic Container Operations/F_VN_FillContainerExp/F_VN_FillContainerExp_TcVnPoint2_LREAL

	{attribute 'TcIecLibraryType'}
	{attribute 'external_name' := 'F_VN_FillContainerExp_TcVnPoint2_LREAL_GUID_AF285AA5_4FF4_4E4A_69E3_0E6DEDEEC01C'}
	(* Partially fill the container with the specified value. Only possible for containers with basic elements. (expert function) *)
	FUNCTION F_VN_FillContainerExp_TcVnPoint2_LREAL : HRESULT
	VAR_INPUT
		ipContainer	:	ITcVnContainer;	(* Container with basic elements *)
		aValue	:	REFERENCE TO TcVnPoint2_LREAL;	(* Value to set the container elements *)
		nStartIdx	:	ULINT;	(* Start index *)
		nCount	:	ULINT;	(* Number of elements to set *)
		hrPrev	:	HRESULT;	(* HRESULT indicating the result of previous operations (If SUCCEEDED(hrPrev) equals false, no operation is executed.) *)
	END_VAR

END_FUNCTION

// Functions/Basic Container Operations/F_VN_FillContainerExp/F_VN_FillContainerExp_TcVnPoint2_REAL

	{attribute 'TcIecLibraryType'}
	{attribute 'external_name' := 'F_VN_FillContainerExp_TcVnPoint2_REAL_GUID_924CF828_952D_4BBF_63CB_CBE3D5AFE8E7'}
	(* Partially fill the container with the specified value. Only possible for containers with basic elements. (expert function) *)
	FUNCTION F_VN_FillContainerExp_TcVnPoint2_REAL : HRESULT
	VAR_INPUT
		ipContainer	:	ITcVnContainer;	(* Container with basic elements *)
		aValue	:	REFERENCE TO TcVnPoint2_REAL;	(* Value to set the container elements *)
		nStartIdx	:	ULINT;	(* Start index *)
		nCount	:	ULINT;	(* Number of elements to set *)
		hrPrev	:	HRESULT;	(* HRESULT indicating the result of previous operations (If SUCCEEDED(hrPrev) equals false, no operation is executed.) *)
	END_VAR

END_FUNCTION

// Functions/Basic Container Operations/F_VN_FillContainerExp/F_VN_FillContainerExp_TcVnPoint3_LREAL

	{attribute 'TcIecLibraryType'}
	{attribute 'external_name' := 'F_VN_FillContainerExp_TcVnPoint3_LREAL_GUID_F7B15BC5_E35E_4D9B_772C_B62DF991F8E2'}
	(* Partially fill the container with the specified value. Only possible for containers with basic elements. (expert function) *)
	FUNCTION F_VN_FillContainerExp_TcVnPoint3_LREAL : HRESULT
	VAR_INPUT
		ipContainer	:	ITcVnContainer;	(* Container with basic elements *)
		aValue	:	REFERENCE TO TcVnPoint3_LREAL;	(* Value to set the container elements *)
		nStartIdx	:	ULINT;	(* Start index *)
		nCount	:	ULINT;	(* Number of elements to set *)
		hrPrev	:	HRESULT;	(* HRESULT indicating the result of previous operations (If SUCCEEDED(hrPrev) equals false, no operation is executed.) *)
	END_VAR

END_FUNCTION

// Functions/Basic Container Operations/F_VN_FillContainerExp/F_VN_FillContainerExp_TcVnPoint3_REAL

	{attribute 'TcIecLibraryType'}
	{attribute 'external_name' := 'F_VN_FillContainerExp_TcVnPoint3_REAL_GUID_2A0D202D_2281_4DA5_7EDB_9B3852C75A24'}
	(* Partially fill the container with the specified value. Only possible for containers with basic elements. (expert function) *)
	FUNCTION F_VN_FillContainerExp_TcVnPoint3_REAL : HRESULT
	VAR_INPUT
		ipContainer	:	ITcVnContainer;	(* Container with basic elements *)
		aValue	:	REFERENCE TO TcVnPoint3_REAL;	(* Value to set the container elements *)
		nStartIdx	:	ULINT;	(* Start index *)
		nCount	:	ULINT;	(* Number of elements to set *)
		hrPrev	:	HRESULT;	(* HRESULT indicating the result of previous operations (If SUCCEEDED(hrPrev) equals false, no operation is executed.) *)
	END_VAR

END_FUNCTION

// Functions/Basic Container Operations/F_VN_FillContainerExp/F_VN_FillContainerExp_TcVnRectangle_DINT

	{attribute 'TcIecLibraryType'}
	{attribute 'external_name' := 'F_VN_FillContainerExp_TcVnRectangle_DINT_GUID_CB65C1C4_7253_4BB7_7951_F3B67396636F'}
	(* Partially fill the container with the specified value. Only possible for containers with basic elements. (expert function) *)
	FUNCTION F_VN_FillContainerExp_TcVnRectangle_DINT : HRESULT
	VAR_INPUT
		ipContainer	:	ITcVnContainer;	(* Container with basic elements *)
		stValue	:	REFERENCE TO TcVnRectangle_DINT;	(* Value to set the container elements *)
		nStartIdx	:	ULINT;	(* Start index *)
		nCount	:	ULINT;	(* Number of elements to set *)
		hrPrev	:	HRESULT;	(* HRESULT indicating the result of previous operations (If SUCCEEDED(hrPrev) equals false, no operation is executed.) *)
	END_VAR

END_FUNCTION

// Functions/Basic Container Operations/F_VN_FillContainerExp/F_VN_FillContainerExp_TcVnVector2_DINT

	{attribute 'TcIecLibraryType'}
	{attribute 'external_name' := 'F_VN_FillContainerExp_TcVnVector2_DINT_GUID_95F7812F_C8CC_4904_6CF5_529EEF1A3A16'}
	(* Partially fill the container with the specified value. Only possible for containers with basic elements. (expert function) *)
	FUNCTION F_VN_FillContainerExp_TcVnVector2_DINT : HRESULT
	VAR_INPUT
		ipContainer	:	ITcVnContainer;	(* Container with basic elements *)
		aValue	:	REFERENCE TO TcVnVector2_DINT;	(* Value to set the container elements *)
		nStartIdx	:	ULINT;	(* Start index *)
		nCount	:	ULINT;	(* Number of elements to set *)
		hrPrev	:	HRESULT;	(* HRESULT indicating the result of previous operations (If SUCCEEDED(hrPrev) equals false, no operation is executed.) *)
	END_VAR

END_FUNCTION

// Functions/Basic Container Operations/F_VN_FillContainerExp/F_VN_FillContainerExp_TcVnVector2_REAL

	{attribute 'TcIecLibraryType'}
	{attribute 'external_name' := 'F_VN_FillContainerExp_TcVnVector2_REAL_GUID_390A06C8_CF35_49F4_5B0A_7E81CA67D63A'}
	(* Partially fill the container with the specified value. Only possible for containers with basic elements. (expert function) *)
	FUNCTION F_VN_FillContainerExp_TcVnVector2_REAL : HRESULT
	VAR_INPUT
		ipContainer	:	ITcVnContainer;	(* Container with basic elements *)
		aValue	:	REFERENCE TO TcVnVector2_REAL;	(* Value to set the container elements *)
		nStartIdx	:	ULINT;	(* Start index *)
		nCount	:	ULINT;	(* Number of elements to set *)
		hrPrev	:	HRESULT;	(* HRESULT indicating the result of previous operations (If SUCCEEDED(hrPrev) equals false, no operation is executed.) *)
	END_VAR

END_FUNCTION

// Functions/Basic Container Operations/F_VN_FillContainerExp/F_VN_FillContainerExp_TcVnVector3_REAL

	{attribute 'TcIecLibraryType'}
	{attribute 'external_name' := 'F_VN_FillContainerExp_TcVnVector3_REAL_GUID_B7C7E24F_49A6_47B2_5FFD_108901EE176E'}
	(* Partially fill the container with the specified value. Only possible for containers with basic elements. (expert function) *)
	FUNCTION F_VN_FillContainerExp_TcVnVector3_REAL : HRESULT
	VAR_INPUT
		ipContainer	:	ITcVnContainer;	(* Container with basic elements *)
		aValue	:	REFERENCE TO TcVnVector3_REAL;	(* Value to set the container elements *)
		nStartIdx	:	ULINT;	(* Start index *)
		nCount	:	ULINT;	(* Number of elements to set *)
		hrPrev	:	HRESULT;	(* HRESULT indicating the result of previous operations (If SUCCEEDED(hrPrev) equals false, no operation is executed.) *)
	END_VAR

END_FUNCTION

// Functions/Basic Container Operations/F_VN_FillContainerExp/F_VN_FillContainerExp_TcVnVector4_DINT

	{attribute 'TcIecLibraryType'}
	{attribute 'external_name' := 'F_VN_FillContainerExp_TcVnVector4_DINT_GUID_906D9A04_C627_4CC2_5283_AF208D3AF31F'}
	(* Partially fill the container with the specified value. Only possible for containers with basic elements. (expert function) *)
	FUNCTION F_VN_FillContainerExp_TcVnVector4_DINT : HRESULT
	VAR_INPUT
		ipContainer	:	ITcVnContainer;	(* Container with basic elements *)
		aValue	:	REFERENCE TO TcVnVector4_DINT;	(* Value to set the container elements *)
		nStartIdx	:	ULINT;	(* Start index *)
		nCount	:	ULINT;	(* Number of elements to set *)
		hrPrev	:	HRESULT;	(* HRESULT indicating the result of previous operations (If SUCCEEDED(hrPrev) equals false, no operation is executed.) *)
	END_VAR

END_FUNCTION

// Functions/Basic Container Operations/F_VN_FillContainerExp/F_VN_FillContainerExp_UDINT

	{attribute 'TcIecLibraryType'}
	{attribute 'external_name' := 'F_VN_FillContainerExp_UDINT_GUID_81507087_988A_481A_58C6_E0C972B957EE'}
	(* Partially fill the container with the specified value. Only possible for containers with basic elements. (expert function) *)
	FUNCTION F_VN_FillContainerExp_UDINT : HRESULT
	VAR_INPUT
		ipContainer	:	ITcVnContainer;	(* Container with basic elements *)
		nValue	:	UDINT;	(* Value to set the container elements *)
		nStartIdx	:	ULINT;	(* Start index *)
		nCount	:	ULINT;	(* Number of elements to set *)
		hrPrev	:	HRESULT;	(* HRESULT indicating the result of previous operations (If SUCCEEDED(hrPrev) equals false, no operation is executed.) *)
	END_VAR

END_FUNCTION

// Functions/Basic Container Operations/F_VN_FillContainerExp/F_VN_FillContainerExp_ULINT

	{attribute 'TcIecLibraryType'}
	{attribute 'external_name' := 'F_VN_FillContainerExp_ULINT_GUID_A18EF9A8_D8CA_4949_591D_AC749B2C5974'}
	(* Partially fill the container with the specified value. Only possible for containers with basic elements. (expert function) *)
	FUNCTION F_VN_FillContainerExp_ULINT : HRESULT
	VAR_INPUT
		ipContainer	:	ITcVnContainer;	(* Container with basic elements *)
		nValue	:	ULINT;	(* Value to set the container elements *)
		nStartIdx	:	ULINT;	(* Start index *)
		nCount	:	ULINT;	(* Number of elements to set *)
		hrPrev	:	HRESULT;	(* HRESULT indicating the result of previous operations (If SUCCEEDED(hrPrev) equals false, no operation is executed.) *)
	END_VAR

END_FUNCTION

// Functions/Basic Container Operations/F_VN_GetAt/F_VN_GetAt_ITcVnContainer

	{attribute 'TcIecLibraryType'}
	{attribute 'external_name' := 'F_VN_GetAt_ITcVnContainer_GUID_44865E92_CAD0_4B4A_4272_4849B4C39D40'}
	(* Gets the ITcVnContainer element at the specified index of the source container. (Alternatively use interface method .GetAt.) *)
	FUNCTION F_VN_GetAt_ITcVnContainer : HRESULT
	VAR_INPUT
		ipSrcContainer	:	ITcVnContainer;	(* Container with ITcVnContainer elements *)
		ipDestContainer	:	REFERENCE TO ITcVnContainer;	(* Returns the container at the specified index *)
		nIndex	:	ULINT;	(* Index of the requested element *)
		hrPrev	:	HRESULT;	(* HRESULT indicating the result of previous operations (If SUCCEEDED(hrPrev) equals false, no operation is executed.) *)
	END_VAR

END_FUNCTION

// Functions/Basic Container Operations/F_VN_GetAt/F_VN_GetAt_LREAL

	{attribute 'TcIecLibraryType'}
	{attribute 'external_name' := 'F_VN_GetAt_LREAL_GUID_9C5E813A_BE30_490B_78C0_A86DA0DDE568'}
	(* Gets the LREAL element at the specified index of the container. *)
	FUNCTION F_VN_GetAt_LREAL : HRESULT
	VAR_INPUT
		ipContainer	:	ITcVnContainer;	(* Container with LREAL elements *)
		fElement	:	REFERENCE TO LREAL;	(* Returns the element at the specified index *)
		nIndex	:	ULINT;	(* Index of the requested element *)
		hrPrev	:	HRESULT;	(* HRESULT indicating the result of previous operations (If SUCCEEDED(hrPrev) equals false, no operation is executed.) *)
	END_VAR

END_FUNCTION

// Functions/Basic Container Operations/F_VN_GetAt/F_VN_GetAt_REAL

	{attribute 'TcIecLibraryType'}
	{attribute 'external_name' := 'F_VN_GetAt_REAL_GUID_5ECF7F87_ED5B_4C04_6E83_7995C54C2B8A'}
	(* Gets the REAL element at the specified index of the container. *)
	FUNCTION F_VN_GetAt_REAL : HRESULT
	VAR_INPUT
		ipContainer	:	ITcVnContainer;	(* Container with REAL elements *)
		fElement	:	REFERENCE TO REAL;	(* Returns the element at the specified index *)
		nIndex	:	ULINT;	(* Index of the requested element *)
		hrPrev	:	HRESULT;	(* HRESULT indicating the result of previous operations (If SUCCEEDED(hrPrev) equals false, no operation is executed.) *)
	END_VAR

END_FUNCTION

// Functions/Basic Container Operations/F_VN_GetAt/F_VN_GetAt_SINT

	{attribute 'TcIecLibraryType'}
	{attribute 'external_name' := 'F_VN_GetAt_SINT_GUID_C8CFAD4B_50AA_4FE9_49EF_8821E0D2F852'}
	(* Gets the SINT element at the specified index of the container. *)
	FUNCTION F_VN_GetAt_SINT : HRESULT
	VAR_INPUT
		ipContainer	:	ITcVnContainer;	(* Container with SINT elements *)
		nElement	:	REFERENCE TO SINT;	(* Returns the element at the specified index *)
		nIndex	:	ULINT;	(* Index of the requested element *)
		hrPrev	:	HRESULT;	(* HRESULT indicating the result of previous operations (If SUCCEEDED(hrPrev) equals false, no operation is executed.) *)
	END_VAR

END_FUNCTION

// Functions/Basic Container Operations/F_VN_GetAt/F_VN_GetAt_TcVnDMatch

	{attribute 'TcIecLibraryType'}
	{attribute 'external_name' := 'F_VN_GetAt_TcVnDMatch_GUID_72DE02D8_2FBB_4A9B_6F20_17D61C75412D'}
	(* Gets the TcVnDMatch element at the specified index of the container. *)
	FUNCTION F_VN_GetAt_TcVnDMatch : HRESULT
	VAR_INPUT
		ipContainer	:	ITcVnContainer;	(* Container with TcVnDMatch elements *)
		stElement	:	REFERENCE TO TcVnDMatch;	(* Returns the element at the specified index *)
		nIndex	:	ULINT;	(* Index of the requested element *)
		hrPrev	:	HRESULT;	(* HRESULT indicating the result of previous operations (If SUCCEEDED(hrPrev) equals false, no operation is executed.) *)
	END_VAR

END_FUNCTION

// Functions/Basic Container Operations/F_VN_GetAt/F_VN_GetAt_TcVnKeyPoint

	{attribute 'TcIecLibraryType'}
	{attribute 'external_name' := 'F_VN_GetAt_TcVnKeyPoint_GUID_6DDCF9E5_53C5_4E89_7350_B8534BE4DE8C'}
	(* Gets the TcVnKeyPoint element at the specified index of the container. *)
	FUNCTION F_VN_GetAt_TcVnKeyPoint : HRESULT
	VAR_INPUT
		ipContainer	:	ITcVnContainer;	(* Container with TcVnKeyPoint elements *)
		stElement	:	REFERENCE TO TcVnKeyPoint;	(* Returns the element at the specified index *)
		nIndex	:	ULINT;	(* Index of the requested element *)
		hrPrev	:	HRESULT;	(* HRESULT indicating the result of previous operations (If SUCCEEDED(hrPrev) equals false, no operation is executed.) *)
	END_VAR

END_FUNCTION

// Functions/Basic Container Operations/F_VN_GetAt/F_VN_GetAt_TcVnPoint2_DINT

	{attribute 'TcIecLibraryType'}
	{attribute 'external_name' := 'F_VN_GetAt_TcVnPoint2_DINT_GUID_A3E7CB2A_186C_4AA5_6A32_E7F1ED1D8F28'}
	(* Gets the TcVnPoint2_DINT element at the specified index of the container. *)
	FUNCTION F_VN_GetAt_TcVnPoint2_DINT : HRESULT
	VAR_INPUT
		ipContainer	:	ITcVnContainer;	(* Container with TcVnPoint2_DINT elements *)
		aElement	:	REFERENCE TO TcVnPoint2_DINT;	(* Returns the element at the specified index *)
		nIndex	:	ULINT;	(* Index of the requested element *)
		hrPrev	:	HRESULT;	(* HRESULT indicating the result of previous operations (If SUCCEEDED(hrPrev) equals false, no operation is executed.) *)
	END_VAR

END_FUNCTION

// Functions/Basic Container Operations/F_VN_GetAt/F_VN_GetAt_TcVnPoint2_LREAL

	{attribute 'TcIecLibraryType'}
	{attribute 'external_name' := 'F_VN_GetAt_TcVnPoint2_LREAL_GUID_DE32B422_1B98_4FBE_485F_B89C695DD92F'}
	(* Gets the TcVnPoint2_LREAL element at the specified index of the container. *)
	FUNCTION F_VN_GetAt_TcVnPoint2_LREAL : HRESULT
	VAR_INPUT
		ipContainer	:	ITcVnContainer;	(* Container with TcVnPoint2_LREAL elements *)
		aElement	:	REFERENCE TO TcVnPoint2_LREAL;	(* Returns the element at the specified index *)
		nIndex	:	ULINT;	(* Index of the requested element *)
		hrPrev	:	HRESULT;	(* HRESULT indicating the result of previous operations (If SUCCEEDED(hrPrev) equals false, no operation is executed.) *)
	END_VAR

END_FUNCTION

// Functions/Basic Container Operations/F_VN_GetAt/F_VN_GetAt_TcVnPoint2_REAL

	{attribute 'TcIecLibraryType'}
	{attribute 'external_name' := 'F_VN_GetAt_TcVnPoint2_REAL_GUID_77C744A6_3021_450F_50EC_1D6178DE094B'}
	(* Gets the TcVnPoint2_REAL element at the specified index of the container. *)
	FUNCTION F_VN_GetAt_TcVnPoint2_REAL : HRESULT
	VAR_INPUT
		ipContainer	:	ITcVnContainer;	(* Container with TcVnPoint2_REAL elements *)
		aElement	:	REFERENCE TO TcVnPoint2_REAL;	(* Returns the element at the specified index *)
		nIndex	:	ULINT;	(* Index of the requested element *)
		hrPrev	:	HRESULT;	(* HRESULT indicating the result of previous operations (If SUCCEEDED(hrPrev) equals false, no operation is executed.) *)
	END_VAR

END_FUNCTION

// Functions/Basic Container Operations/F_VN_GetAt/F_VN_GetAt_TcVnPoint3_LREAL

	{attribute 'TcIecLibraryType'}
	{attribute 'external_name' := 'F_VN_GetAt_TcVnPoint3_LREAL_GUID_D0E0E7BC_622F_41A3_7EAA_2EC3215206B1'}
	(* Gets the TcVnPoint3_LREAL element at the specified index of the container. *)
	FUNCTION F_VN_GetAt_TcVnPoint3_LREAL : HRESULT
	VAR_INPUT
		ipContainer	:	ITcVnContainer;	(* Container with TcVnPoint3_LREAL elements *)
		aElement	:	REFERENCE TO TcVnPoint3_LREAL;	(* Returns the element at the specified index *)
		nIndex	:	ULINT;	(* Index of the requested element *)
		hrPrev	:	HRESULT;	(* HRESULT indicating the result of previous operations (If SUCCEEDED(hrPrev) equals false, no operation is executed.) *)
	END_VAR

END_FUNCTION

// Functions/Basic Container Operations/F_VN_GetAt/F_VN_GetAt_TcVnPoint3_REAL

	{attribute 'TcIecLibraryType'}
	{attribute 'external_name' := 'F_VN_GetAt_TcVnPoint3_REAL_GUID_4A8425D2_2136_4B6B_6A35_81E6A6B2C299'}
	(* Gets the TcVnPoint3_REAL element at the specified index of the container. *)
	FUNCTION F_VN_GetAt_TcVnPoint3_REAL : HRESULT
	VAR_INPUT
		ipContainer	:	ITcVnContainer;	(* Container with TcVnPoint3_REAL elements *)
		aElement	:	REFERENCE TO TcVnPoint3_REAL;	(* Returns the element at the specified index *)
		nIndex	:	ULINT;	(* Index of the requested element *)
		hrPrev	:	HRESULT;	(* HRESULT indicating the result of previous operations (If SUCCEEDED(hrPrev) equals false, no operation is executed.) *)
	END_VAR

END_FUNCTION

// Functions/Basic Container Operations/F_VN_GetAt/F_VN_GetAt_TcVnRectangle_DINT

	{attribute 'TcIecLibraryType'}
	{attribute 'external_name' := 'F_VN_GetAt_TcVnRectangle_DINT_GUID_356AAAF8_B754_4C6D_6C6C_03583DAF9A88'}
	(* Gets the TcVnRectangle_DINT element at the specified index of the container. *)
	FUNCTION F_VN_GetAt_TcVnRectangle_DINT : HRESULT
	VAR_INPUT
		ipContainer	:	ITcVnContainer;	(* Container with TcVnRectangle_DINT elements *)
		stElement	:	REFERENCE TO TcVnRectangle_DINT;	(* Returns the element at the specified index *)
		nIndex	:	ULINT;	(* Index of the requested element *)
		hrPrev	:	HRESULT;	(* HRESULT indicating the result of previous operations (If SUCCEEDED(hrPrev) equals false, no operation is executed.) *)
	END_VAR

END_FUNCTION

// Functions/Basic Container Operations/F_VN_GetAt/F_VN_GetAt_TcVnVector2_DINT

	{attribute 'TcIecLibraryType'}
	{attribute 'external_name' := 'F_VN_GetAt_TcVnVector2_DINT_GUID_A71B58C0_6650_470A_4444_319FEF2C83A0'}
	(* Gets the TcVnVector2_DINT element at the specified index of the container. *)
	FUNCTION F_VN_GetAt_TcVnVector2_DINT : HRESULT
	VAR_INPUT
		ipContainer	:	ITcVnContainer;	(* Container with TcVnVector2_DINT elements *)
		aElement	:	REFERENCE TO TcVnVector2_DINT;	(* Returns the element at the specified index *)
		nIndex	:	ULINT;	(* Index of the requested element *)
		hrPrev	:	HRESULT;	(* HRESULT indicating the result of previous operations (If SUCCEEDED(hrPrev) equals false, no operation is executed.) *)
	END_VAR

END_FUNCTION

// Functions/Basic Container Operations/F_VN_GetAt/F_VN_GetAt_TcVnVector2_REAL

	{attribute 'TcIecLibraryType'}
	{attribute 'external_name' := 'F_VN_GetAt_TcVnVector2_REAL_GUID_D396E14D_EF3F_4F4A_4C6D_44BBF627B321'}
	(* Gets the TcVnVector2_REAL element at the specified index of the container. *)
	FUNCTION F_VN_GetAt_TcVnVector2_REAL : HRESULT
	VAR_INPUT
		ipContainer	:	ITcVnContainer;	(* Container with TcVnVector2_REAL elements *)
		aElement	:	REFERENCE TO TcVnVector2_REAL;	(* Returns the element at the specified index *)
		nIndex	:	ULINT;	(* Index of the requested element *)
		hrPrev	:	HRESULT;	(* HRESULT indicating the result of previous operations (If SUCCEEDED(hrPrev) equals false, no operation is executed.) *)
	END_VAR

END_FUNCTION

// Functions/Basic Container Operations/F_VN_GetAt/F_VN_GetAt_TcVnVector3_REAL

	{attribute 'TcIecLibraryType'}
	{attribute 'external_name' := 'F_VN_GetAt_TcVnVector3_REAL_GUID_AF81D7C4_31B9_4A01_73A2_63C9B3546329'}
	(* Gets the TcVnVector3_REAL element at the specified index of the container. *)
	FUNCTION F_VN_GetAt_TcVnVector3_REAL : HRESULT
	VAR_INPUT
		ipContainer	:	ITcVnContainer;	(* Container with TcVnVector3_REAL elements *)
		aElement	:	REFERENCE TO TcVnVector3_REAL;	(* Returns the element at the specified index *)
		nIndex	:	ULINT;	(* Index of the requested element *)
		hrPrev	:	HRESULT;	(* HRESULT indicating the result of previous operations (If SUCCEEDED(hrPrev) equals false, no operation is executed.) *)
	END_VAR

END_FUNCTION

// Functions/Basic Container Operations/F_VN_GetAt/F_VN_GetAt_TcVnVector4_DINT

	{attribute 'TcIecLibraryType'}
	{attribute 'external_name' := 'F_VN_GetAt_TcVnVector4_DINT_GUID_AAD69F4C_C07F_48F6_4349_435D928F282B'}
	(* Gets the TcVnVector4_DINT element at the specified index of the container. *)
	FUNCTION F_VN_GetAt_TcVnVector4_DINT : HRESULT
	VAR_INPUT
		ipContainer	:	ITcVnContainer;	(* Container with TcVnVector4_DINT elements *)
		aElement	:	REFERENCE TO TcVnVector4_DINT;	(* Returns the element at the specified index *)
		nIndex	:	ULINT;	(* Index of the requested element *)
		hrPrev	:	HRESULT;	(* HRESULT indicating the result of previous operations (If SUCCEEDED(hrPrev) equals false, no operation is executed.) *)
	END_VAR

END_FUNCTION

// Functions/Basic Container Operations/F_VN_GetAt/F_VN_GetAt_UDINT

	{attribute 'TcIecLibraryType'}
	{attribute 'external_name' := 'F_VN_GetAt_UDINT_GUID_188CFCA2_76FC_48C3_75F7_28682C8DF1EA'}
	(* Gets the UDINT element at the specified index of the container. *)
	FUNCTION F_VN_GetAt_UDINT : HRESULT
	VAR_INPUT
		ipContainer	:	ITcVnContainer;	(* Container with UDINT elements *)
		nElement	:	REFERENCE TO UDINT;	(* Returns the element at the specified index *)
		nIndex	:	ULINT;	(* Index of the requested element *)
		hrPrev	:	HRESULT;	(* HRESULT indicating the result of previous operations (If SUCCEEDED(hrPrev) equals false, no operation is executed.) *)
	END_VAR

END_FUNCTION

// Functions/Basic Container Operations/F_VN_GetAt/F_VN_GetAt_ULINT

	{attribute 'TcIecLibraryType'}
	{attribute 'external_name' := 'F_VN_GetAt_ULINT_GUID_1BAB2A71_FF27_4594_7432_F808C4507CFB'}
	(* Gets the ULINT element at the specified index of the container. *)
	FUNCTION F_VN_GetAt_ULINT : HRESULT
	VAR_INPUT
		ipContainer	:	ITcVnContainer;	(* Container with ULINT elements *)
		nElement	:	REFERENCE TO ULINT;	(* Returns the element at the specified index *)
		nIndex	:	ULINT;	(* Index of the requested element *)
		hrPrev	:	HRESULT;	(* HRESULT indicating the result of previous operations (If SUCCEEDED(hrPrev) equals false, no operation is executed.) *)
	END_VAR

END_FUNCTION

// Functions/Basic Container Operations/F_VN_InsertIntoContainer/F_VN_InsertIntoContainer_ITcVnContainer

	{attribute 'TcIecLibraryType'}
	{attribute 'external_name' := 'F_VN_InsertIntoContainer_ITcVnContainer_GUID_0110B084_B56F_4891_4675_B8D488AFC718'}
	(* Insert an element (or a range of elements) into a container before the specified position. *)
	FUNCTION F_VN_InsertIntoContainer_ITcVnContainer : HRESULT
	VAR_INPUT
		ipElement	:	ITcVnContainer;	(* Single element to insert into ipContainer or container with several elements *)
		ipContainer	:	ITcVnContainer;	(* Container in which to insert the element *)
		nIndex	:	ULINT;	(* Position, before which the element will be inserted *)
		hrPrev	:	HRESULT;	(* HRESULT indicating the result of previous operations (If SUCCEEDED(hrPrev) equals false, no operation is executed.) *)
	END_VAR

END_FUNCTION

// Functions/Basic Container Operations/F_VN_InsertIntoContainer/F_VN_InsertIntoContainer_ITcVnForwardIterator

	{attribute 'TcIecLibraryType'}
	{attribute 'external_name' := 'F_VN_InsertIntoContainer_ITcVnForwardIterator_GUID_5C6E5723_E67A_4E33_425A_4DCDC390871B'}
	(* Insert an element (represented by an iterator) into a container before the specified position. *)
	FUNCTION F_VN_InsertIntoContainer_ITcVnForwardIterator : HRESULT
	VAR_INPUT
		ipElement	:	ITcVnForwardIterator;	(* Single element to insert into ipContainer *)
		ipContainer	:	ITcVnContainer;	(* Container in which to insert the element *)
		nIndex	:	ULINT;	(* Position, before which the element will be inserted *)
		hrPrev	:	HRESULT;	(* HRESULT indicating the result of previous operations (If SUCCEEDED(hrPrev) equals false, no operation is executed.) *)
	END_VAR

END_FUNCTION

// Functions/Basic Container Operations/F_VN_InsertIntoContainer/F_VN_InsertIntoContainer_LREAL

	{attribute 'TcIecLibraryType'}
	{attribute 'external_name' := 'F_VN_InsertIntoContainer_LREAL_GUID_AE743BEA_6E87_4AE5_4E59_3844A25FC8E3'}
	(* Insert an element of type LREAL into a container before the specified position. *)
	FUNCTION F_VN_InsertIntoContainer_LREAL : HRESULT
	VAR_INPUT
		fElement	:	LREAL;	(* Single element to insert into ipContainer *)
		ipContainer	:	ITcVnContainer;	(* Container in which to insert the element *)
		nIndex	:	ULINT;	(* Position, before which the element will be inserted *)
		hrPrev	:	HRESULT;	(* HRESULT indicating the result of previous operations (If SUCCEEDED(hrPrev) equals false, no operation is executed.) *)
	END_VAR

END_FUNCTION

// Functions/Basic Container Operations/F_VN_InsertIntoContainer/F_VN_InsertIntoContainer_REAL

	{attribute 'TcIecLibraryType'}
	{attribute 'external_name' := 'F_VN_InsertIntoContainer_REAL_GUID_E26AED07_9C37_4B3A_5A42_56372835AC35'}
	(* Insert an element of type REAL into a container before the specified position. *)
	FUNCTION F_VN_InsertIntoContainer_REAL : HRESULT
	VAR_INPUT
		fElement	:	REAL;	(* Single element to insert into ipContainer *)
		ipContainer	:	ITcVnContainer;	(* Container in which to insert the element *)
		nIndex	:	ULINT;	(* Position, before which the element will be inserted *)
		hrPrev	:	HRESULT;	(* HRESULT indicating the result of previous operations (If SUCCEEDED(hrPrev) equals false, no operation is executed.) *)
	END_VAR

END_FUNCTION

// Functions/Basic Container Operations/F_VN_InsertIntoContainer/F_VN_InsertIntoContainer_SINT

	{attribute 'TcIecLibraryType'}
	{attribute 'external_name' := 'F_VN_InsertIntoContainer_SINT_GUID_00E43975_0F52_4C51_54A1_902F3C1CA547'}
	(* Insert an element of type SINT into a container before the specified position. *)
	FUNCTION F_VN_InsertIntoContainer_SINT : HRESULT
	VAR_INPUT
		nElement	:	SINT;	(* Single element to insert into ipContainer *)
		ipContainer	:	ITcVnContainer;	(* Container in which to insert the element *)
		nIndex	:	ULINT;	(* Position, before which the element will be inserted *)
		hrPrev	:	HRESULT;	(* HRESULT indicating the result of previous operations (If SUCCEEDED(hrPrev) equals false, no operation is executed.) *)
	END_VAR

END_FUNCTION

// Functions/Basic Container Operations/F_VN_InsertIntoContainer/F_VN_InsertIntoContainer_TcVnDMatch

	{attribute 'TcIecLibraryType'}
	{attribute 'external_name' := 'F_VN_InsertIntoContainer_TcVnDMatch_GUID_BE44CCFA_1D20_430A_723F_107DE80A627D'}
	(* Insert an element of type TcVnDMatch into a container before the specified position. *)
	FUNCTION F_VN_InsertIntoContainer_TcVnDMatch : HRESULT
	VAR_INPUT
		stElement	:	REFERENCE TO TcVnDMatch;	(* Single element to insert into ipContainer *)
		ipContainer	:	ITcVnContainer;	(* Container in which to insert the element *)
		nIndex	:	ULINT;	(* Position, before which the element will be inserted *)
		hrPrev	:	HRESULT;	(* HRESULT indicating the result of previous operations (If SUCCEEDED(hrPrev) equals false, no operation is executed.) *)
	END_VAR

END_FUNCTION

// Functions/Basic Container Operations/F_VN_InsertIntoContainer/F_VN_InsertIntoContainer_TcVnKeyPoint

	{attribute 'TcIecLibraryType'}
	{attribute 'external_name' := 'F_VN_InsertIntoContainer_TcVnKeyPoint_GUID_6AE81B79_DF4B_4EAE_7FD5_E6ACF8A9FD13'}
	(* Insert an element of type TcVnKeyPoint into a container before the specified position. *)
	FUNCTION F_VN_InsertIntoContainer_TcVnKeyPoint : HRESULT
	VAR_INPUT
		stElement	:	REFERENCE TO TcVnKeyPoint;	(* Single element to insert into ipContainer *)
		ipContainer	:	ITcVnContainer;	(* Container in which to insert the element *)
		nIndex	:	ULINT;	(* Position, before which the element will be inserted *)
		hrPrev	:	HRESULT;	(* HRESULT indicating the result of previous operations (If SUCCEEDED(hrPrev) equals false, no operation is executed.) *)
	END_VAR

END_FUNCTION

// Functions/Basic Container Operations/F_VN_InsertIntoContainer/F_VN_InsertIntoContainer_TcVnPoint2_DINT

	{attribute 'TcIecLibraryType'}
	{attribute 'external_name' := 'F_VN_InsertIntoContainer_TcVnPoint2_DINT_GUID_2985E9B6_E0C8_483F_6BE6_3210B315F8ED'}
	(* Insert an element of type TcVnPoint2_DINT into a container before the specified position. *)
	FUNCTION F_VN_InsertIntoContainer_TcVnPoint2_DINT : HRESULT
	VAR_INPUT
		aElement	:	REFERENCE TO TcVnPoint2_DINT;	(* Single element to insert into ipContainer *)
		ipContainer	:	ITcVnContainer;	(* Container in which to insert the element *)
		nIndex	:	ULINT;	(* Position, before which the element will be inserted *)
		hrPrev	:	HRESULT;	(* HRESULT indicating the result of previous operations (If SUCCEEDED(hrPrev) equals false, no operation is executed.) *)
	END_VAR

END_FUNCTION

// Functions/Basic Container Operations/F_VN_InsertIntoContainer/F_VN_InsertIntoContainer_TcVnPoint2_LREAL

	{attribute 'TcIecLibraryType'}
	{attribute 'external_name' := 'F_VN_InsertIntoContainer_TcVnPoint2_LREAL_GUID_D3FE8241_C89F_4217_7D37_04980971245F'}
	(* Insert an element of type TcVnPoint2_LREAL into a container before the specified position. *)
	FUNCTION F_VN_InsertIntoContainer_TcVnPoint2_LREAL : HRESULT
	VAR_INPUT
		aElement	:	REFERENCE TO TcVnPoint2_LREAL;	(* Single element to insert into ipContainer *)
		ipContainer	:	ITcVnContainer;	(* Container in which to insert the element *)
		nIndex	:	ULINT;	(* Position, before which the element will be inserted *)
		hrPrev	:	HRESULT;	(* HRESULT indicating the result of previous operations (If SUCCEEDED(hrPrev) equals false, no operation is executed.) *)
	END_VAR

END_FUNCTION

// Functions/Basic Container Operations/F_VN_InsertIntoContainer/F_VN_InsertIntoContainer_TcVnPoint2_REAL

	{attribute 'TcIecLibraryType'}
	{attribute 'external_name' := 'F_VN_InsertIntoContainer_TcVnPoint2_REAL_GUID_AEB39457_9744_4A94_56D3_B616F60B5FED'}
	(* Insert an element of type TcVnPoint2_REAL into a container before the specified position. *)
	FUNCTION F_VN_InsertIntoContainer_TcVnPoint2_REAL : HRESULT
	VAR_INPUT
		aElement	:	REFERENCE TO TcVnPoint2_REAL;	(* Single element to insert into ipContainer *)
		ipContainer	:	ITcVnContainer;	(* Container in which to insert the element *)
		nIndex	:	ULINT;	(* Position, before which the element will be inserted *)
		hrPrev	:	HRESULT;	(* HRESULT indicating the result of previous operations (If SUCCEEDED(hrPrev) equals false, no operation is executed.) *)
	END_VAR

END_FUNCTION

// Functions/Basic Container Operations/F_VN_InsertIntoContainer/F_VN_InsertIntoContainer_TcVnPoint3_LREAL

	{attribute 'TcIecLibraryType'}
	{attribute 'external_name' := 'F_VN_InsertIntoContainer_TcVnPoint3_LREAL_GUID_DBBF519F_ECC3_4286_5B9C_7CB45315FBBD'}
	(* Insert an element of type TcVnPoint3_LREAL into a container before the specified position. *)
	FUNCTION F_VN_InsertIntoContainer_TcVnPoint3_LREAL : HRESULT
	VAR_INPUT
		aElement	:	REFERENCE TO TcVnPoint3_LREAL;	(* Single element to insert into ipContainer *)
		ipContainer	:	ITcVnContainer;	(* Container in which to insert the element *)
		nIndex	:	ULINT;	(* Position, before which the element will be inserted *)
		hrPrev	:	HRESULT;	(* HRESULT indicating the result of previous operations (If SUCCEEDED(hrPrev) equals false, no operation is executed.) *)
	END_VAR

END_FUNCTION

// Functions/Basic Container Operations/F_VN_InsertIntoContainer/F_VN_InsertIntoContainer_TcVnPoint3_REAL

	{attribute 'TcIecLibraryType'}
	{attribute 'external_name' := 'F_VN_InsertIntoContainer_TcVnPoint3_REAL_GUID_BAAF1C0A_D5E1_4C0D_7F9A_B1C06909395B'}
	(* Insert an element of type TcVnPoint3_REAL into a container before the specified position. *)
	FUNCTION F_VN_InsertIntoContainer_TcVnPoint3_REAL : HRESULT
	VAR_INPUT
		aElement	:	REFERENCE TO TcVnPoint3_REAL;	(* Single element to insert into ipContainer *)
		ipContainer	:	ITcVnContainer;	(* Container in which to insert the element *)
		nIndex	:	ULINT;	(* Position, before which the element will be inserted *)
		hrPrev	:	HRESULT;	(* HRESULT indicating the result of previous operations (If SUCCEEDED(hrPrev) equals false, no operation is executed.) *)
	END_VAR

END_FUNCTION

// Functions/Basic Container Operations/F_VN_InsertIntoContainer/F_VN_InsertIntoContainer_TcVnRectangle_DINT

	{attribute 'TcIecLibraryType'}
	{attribute 'external_name' := 'F_VN_InsertIntoContainer_TcVnRectangle_DINT_GUID_B1F044D9_26D1_4253_4735_F5473B720FC3'}
	(* Insert an element of type TcVnRectangle_DINT into a container before the specified position. *)
	FUNCTION F_VN_InsertIntoContainer_TcVnRectangle_DINT : HRESULT
	VAR_INPUT
		stElement	:	REFERENCE TO TcVnRectangle_DINT;	(* Single element to insert into ipContainer *)
		ipContainer	:	ITcVnContainer;	(* Container in which to insert the element *)
		nIndex	:	ULINT;	(* Position, before which the element will be inserted *)
		hrPrev	:	HRESULT;	(* HRESULT indicating the result of previous operations (If SUCCEEDED(hrPrev) equals false, no operation is executed.) *)
	END_VAR

END_FUNCTION

// Functions/Basic Container Operations/F_VN_InsertIntoContainer/F_VN_InsertIntoContainer_TcVnVector2_DINT

	{attribute 'TcIecLibraryType'}
	{attribute 'external_name' := 'F_VN_InsertIntoContainer_TcVnVector2_DINT_GUID_4A1F1FD8_6202_431D_4276_39EB5F4B408D'}
	(* Insert an element of type TcVnVector2_DINT into a container before the specified position. *)
	FUNCTION F_VN_InsertIntoContainer_TcVnVector2_DINT : HRESULT
	VAR_INPUT
		aElement	:	REFERENCE TO TcVnVector2_DINT;	(* Single element to insert into ipContainer *)
		ipContainer	:	ITcVnContainer;	(* Container in which to insert the element *)
		nIndex	:	ULINT;	(* Position, before which the element will be inserted *)
		hrPrev	:	HRESULT;	(* HRESULT indicating the result of previous operations (If SUCCEEDED(hrPrev) equals false, no operation is executed.) *)
	END_VAR

END_FUNCTION

// Functions/Basic Container Operations/F_VN_InsertIntoContainer/F_VN_InsertIntoContainer_TcVnVector2_REAL

	{attribute 'TcIecLibraryType'}
	{attribute 'external_name' := 'F_VN_InsertIntoContainer_TcVnVector2_REAL_GUID_3B8D37AE_FC29_4497_5526_E776BB5983F8'}
	(* Insert an element of type TcVnVector2_REAL into a container before the specified position. *)
	FUNCTION F_VN_InsertIntoContainer_TcVnVector2_REAL : HRESULT
	VAR_INPUT
		aElement	:	REFERENCE TO TcVnVector2_REAL;	(* Single element to insert into ipContainer *)
		ipContainer	:	ITcVnContainer;	(* Container in which to insert the element *)
		nIndex	:	ULINT;	(* Position, before which the element will be inserted *)
		hrPrev	:	HRESULT;	(* HRESULT indicating the result of previous operations (If SUCCEEDED(hrPrev) equals false, no operation is executed.) *)
	END_VAR

END_FUNCTION

// Functions/Basic Container Operations/F_VN_InsertIntoContainer/F_VN_InsertIntoContainer_TcVnVector3_REAL

	{attribute 'TcIecLibraryType'}
	{attribute 'external_name' := 'F_VN_InsertIntoContainer_TcVnVector3_REAL_GUID_A2DD18C3_5ED0_4727_4E53_153C77587D18'}
	(* Insert an element of type TcVnVector3_REAL into a container before the specified position. *)
	FUNCTION F_VN_InsertIntoContainer_TcVnVector3_REAL : HRESULT
	VAR_INPUT
		aElement	:	REFERENCE TO TcVnVector3_REAL;	(* Single element to insert into ipContainer *)
		ipContainer	:	ITcVnContainer;	(* Container in which to insert the element *)
		nIndex	:	ULINT;	(* Position, before which the element will be inserted *)
		hrPrev	:	HRESULT;	(* HRESULT indicating the result of previous operations (If SUCCEEDED(hrPrev) equals false, no operation is executed.) *)
	END_VAR

END_FUNCTION

// Functions/Basic Container Operations/F_VN_InsertIntoContainer/F_VN_InsertIntoContainer_TcVnVector4_DINT

	{attribute 'TcIecLibraryType'}
	{attribute 'external_name' := 'F_VN_InsertIntoContainer_TcVnVector4_DINT_GUID_96F6F060_65D8_4371_7EAC_79DB09AD2300'}
	(* Insert an element of type TcVnVector4_DINT into a container before the specified position. *)
	FUNCTION F_VN_InsertIntoContainer_TcVnVector4_DINT : HRESULT
	VAR_INPUT
		aElement	:	REFERENCE TO TcVnVector4_DINT;	(* Single element to insert into ipContainer *)
		ipContainer	:	ITcVnContainer;	(* Container in which to insert the element *)
		nIndex	:	ULINT;	(* Position, before which the element will be inserted *)
		hrPrev	:	HRESULT;	(* HRESULT indicating the result of previous operations (If SUCCEEDED(hrPrev) equals false, no operation is executed.) *)
	END_VAR

END_FUNCTION

// Functions/Basic Container Operations/F_VN_InsertIntoContainer/F_VN_InsertIntoContainer_UDINT

	{attribute 'TcIecLibraryType'}
	{attribute 'external_name' := 'F_VN_InsertIntoContainer_UDINT_GUID_6A1DC1FD_9D9A_4F2B_7E6E_4BB54EA44066'}
	(* Insert an element of type UDINT into a container before the specified position. *)
	FUNCTION F_VN_InsertIntoContainer_UDINT : HRESULT
	VAR_INPUT
		nElement	:	UDINT;	(* Single element to insert into ipContainer *)
		ipContainer	:	ITcVnContainer;	(* Container in which to insert the element *)
		nIndex	:	ULINT;	(* Position, before which the element will be inserted *)
		hrPrev	:	HRESULT;	(* HRESULT indicating the result of previous operations (If SUCCEEDED(hrPrev) equals false, no operation is executed.) *)
	END_VAR

END_FUNCTION

// Functions/Basic Container Operations/F_VN_InsertIntoContainer/F_VN_InsertIntoContainer_ULINT

	{attribute 'TcIecLibraryType'}
	{attribute 'external_name' := 'F_VN_InsertIntoContainer_ULINT_GUID_D164A892_311E_4E8A_7C71_1C565A95E796'}
	(* Insert an element of type ULINT into a container before the specified position. *)
	FUNCTION F_VN_InsertIntoContainer_ULINT : HRESULT
	VAR_INPUT
		nElement	:	ULINT;	(* Single element to insert into ipContainer *)
		ipContainer	:	ITcVnContainer;	(* Container in which to insert the element *)
		nIndex	:	ULINT;	(* Position, before which the element will be inserted *)
		hrPrev	:	HRESULT;	(* HRESULT indicating the result of previous operations (If SUCCEEDED(hrPrev) equals false, no operation is executed.) *)
	END_VAR

END_FUNCTION

// Functions/Basic Container Operations/F_VN_SetAt/F_VN_SetAt_ITcVnContainer

	{attribute 'TcIecLibraryType'}
	{attribute 'external_name' := 'F_VN_SetAt_ITcVnContainer_GUID_9BAEB5B9_B210_4701_4D57_000E6AE0D226'}
	(* Sets the element at the specified index of the container. (Alternatively use interface method .SetAt.) *)
	FUNCTION F_VN_SetAt_ITcVnContainer : HRESULT
	VAR_INPUT
		ipElement	:	ITcVnContainer;	(* Element to set at the specified container position *)
		ipContainer	:	ITcVnContainer;	(* Container with ITcVnContainer elements, in which the element at position nIndex is replaced by ipElement *)
		nIndex	:	ULINT;	(* Index *)
		hrPrev	:	HRESULT;	(* HRESULT indicating the result of previous operations (If SUCCEEDED(hrPrev) equals false, no operation is executed.) *)
	END_VAR

END_FUNCTION

// Functions/Basic Container Operations/F_VN_SetAt/F_VN_SetAt_LREAL

	{attribute 'TcIecLibraryType'}
	{attribute 'external_name' := 'F_VN_SetAt_LREAL_GUID_9EFA71CF_3B87_433E_7127_018DECBE5651'}
	(* Sets the element at the specified index of the container. *)
	FUNCTION F_VN_SetAt_LREAL : HRESULT
	VAR_INPUT
		fElement	:	LREAL;	(* Element to set at the specified container position *)
		ipContainer	:	ITcVnContainer;	(* Container with LREAL elements, in which the element at position nIndex is replaced by fElement *)
		nIndex	:	ULINT;	(* Index *)
		hrPrev	:	HRESULT;	(* HRESULT indicating the result of previous operations (If SUCCEEDED(hrPrev) equals false, no operation is executed.) *)
	END_VAR

END_FUNCTION

// Functions/Basic Container Operations/F_VN_SetAt/F_VN_SetAt_REAL

	{attribute 'TcIecLibraryType'}
	{attribute 'external_name' := 'F_VN_SetAt_REAL_GUID_51ECAF3A_275E_4F50_645E_DF0A48169BCD'}
	(* Sets the element at the specified index of the container. *)
	FUNCTION F_VN_SetAt_REAL : HRESULT
	VAR_INPUT
		fElement	:	REAL;	(* Element to set at the specified container position *)
		ipContainer	:	ITcVnContainer;	(* Container with REAL elements, in which the element at position nIndex is replaced by fElement *)
		nIndex	:	ULINT;	(* Index *)
		hrPrev	:	HRESULT;	(* HRESULT indicating the result of previous operations (If SUCCEEDED(hrPrev) equals false, no operation is executed.) *)
	END_VAR

END_FUNCTION

// Functions/Basic Container Operations/F_VN_SetAt/F_VN_SetAt_SINT

	{attribute 'TcIecLibraryType'}
	{attribute 'external_name' := 'F_VN_SetAt_SINT_GUID_8F305128_B33D_4EFC_4CBD_41B4443A2F77'}
	(* Sets the element at the specified index of the container. *)
	FUNCTION F_VN_SetAt_SINT : HRESULT
	VAR_INPUT
		nElement	:	SINT;	(* Element to set at the specified container position *)
		ipContainer	:	ITcVnContainer;	(* Container with SINT elements, in which the element at position nIndex is replaced by nElement *)
		nIndex	:	ULINT;	(* Index *)
		hrPrev	:	HRESULT;	(* HRESULT indicating the result of previous operations (If SUCCEEDED(hrPrev) equals false, no operation is executed.) *)
	END_VAR

END_FUNCTION

// Functions/Basic Container Operations/F_VN_SetAt/F_VN_SetAt_TcVnDMatch

	{attribute 'TcIecLibraryType'}
	{attribute 'external_name' := 'F_VN_SetAt_TcVnDMatch_GUID_02AF53D8_31D9_49EA_545E_14AC9A4E6650'}
	(* Sets the element at the specified index of the container. *)
	FUNCTION F_VN_SetAt_TcVnDMatch : HRESULT
	VAR_INPUT
		stElement	:	REFERENCE TO TcVnDMatch;	(* Element to set at the specified container position *)
		ipContainer	:	ITcVnContainer;	(* Container with TcVnDMatch elements, in which the element at position nIndex is replaced by stElement *)
		nIndex	:	ULINT;	(* Index *)
		hrPrev	:	HRESULT;	(* HRESULT indicating the result of previous operations (If SUCCEEDED(hrPrev) equals false, no operation is executed.) *)
	END_VAR

END_FUNCTION

// Functions/Basic Container Operations/F_VN_SetAt/F_VN_SetAt_TcVnKeyPoint

	{attribute 'TcIecLibraryType'}
	{attribute 'external_name' := 'F_VN_SetAt_TcVnKeyPoint_GUID_7A3B6170_C08B_45A2_4FFC_46162E6FCBCC'}
	(* Sets the element at the specified index of the container. *)
	FUNCTION F_VN_SetAt_TcVnKeyPoint : HRESULT
	VAR_INPUT
		stElement	:	REFERENCE TO TcVnKeyPoint;	(* Element to set at the specified container position *)
		ipContainer	:	ITcVnContainer;	(* Container with TcVnKeyPoint elements, in which the element at position nIndex is replaced by stElement *)
		nIndex	:	ULINT;	(* Index *)
		hrPrev	:	HRESULT;	(* HRESULT indicating the result of previous operations (If SUCCEEDED(hrPrev) equals false, no operation is executed.) *)
	END_VAR

END_FUNCTION

// Functions/Basic Container Operations/F_VN_SetAt/F_VN_SetAt_TcVnPoint2_DINT

	{attribute 'TcIecLibraryType'}
	{attribute 'external_name' := 'F_VN_SetAt_TcVnPoint2_DINT_GUID_1775E978_1D8A_4976_7141_1F6D7905A244'}
	(* Sets the element at the specified index of the container. *)
	FUNCTION F_VN_SetAt_TcVnPoint2_DINT : HRESULT
	VAR_INPUT
		aElement	:	REFERENCE TO TcVnPoint2_DINT;	(* Element to set at the specified container position *)
		ipContainer	:	ITcVnContainer;	(* Container with TcVnPoint2_DINT elements, in which the element at position nIndex is replaced by aElement *)
		nIndex	:	ULINT;	(* Index *)
		hrPrev	:	HRESULT;	(* HRESULT indicating the result of previous operations (If SUCCEEDED(hrPrev) equals false, no operation is executed.) *)
	END_VAR

END_FUNCTION

// Functions/Basic Container Operations/F_VN_SetAt/F_VN_SetAt_TcVnPoint2_LREAL

	{attribute 'TcIecLibraryType'}
	{attribute 'external_name' := 'F_VN_SetAt_TcVnPoint2_LREAL_GUID_1C4C1C4D_5B66_4A17_693B_A37B7D454C8B'}
	(* Sets the element at the specified index of the container. *)
	FUNCTION F_VN_SetAt_TcVnPoint2_LREAL : HRESULT
	VAR_INPUT
		aElement	:	REFERENCE TO TcVnPoint2_LREAL;	(* Element to set at the specified container position *)
		ipContainer	:	ITcVnContainer;	(* Container with TcVnPoint2_LREAL elements, in which the element at position nIndex is replaced by aElement *)
		nIndex	:	ULINT;	(* Index *)
		hrPrev	:	HRESULT;	(* HRESULT indicating the result of previous operations (If SUCCEEDED(hrPrev) equals false, no operation is executed.) *)
	END_VAR

END_FUNCTION

// Functions/Basic Container Operations/F_VN_SetAt/F_VN_SetAt_TcVnPoint2_REAL

	{attribute 'TcIecLibraryType'}
	{attribute 'external_name' := 'F_VN_SetAt_TcVnPoint2_REAL_GUID_4C4584D3_E981_4652_52E3_C1625698817B'}
	(* Sets the element at the specified index of the container. *)
	FUNCTION F_VN_SetAt_TcVnPoint2_REAL : HRESULT
	VAR_INPUT
		aElement	:	REFERENCE TO TcVnPoint2_REAL;	(* Element to set at the specified container position *)
		ipContainer	:	ITcVnContainer;	(* Container with TcVnPoint2_REAL elements, in which the element at position nIndex is replaced by aElement *)
		nIndex	:	ULINT;	(* Index *)
		hrPrev	:	HRESULT;	(* HRESULT indicating the result of previous operations (If SUCCEEDED(hrPrev) equals false, no operation is executed.) *)
	END_VAR

END_FUNCTION

// Functions/Basic Container Operations/F_VN_SetAt/F_VN_SetAt_TcVnPoint3_LREAL

	{attribute 'TcIecLibraryType'}
	{attribute 'external_name' := 'F_VN_SetAt_TcVnPoint3_LREAL_GUID_D57FA1C2_AC16_4B48_5A76_F05E823BFA97'}
	(* Sets the element at the specified index of the container. *)
	FUNCTION F_VN_SetAt_TcVnPoint3_LREAL : HRESULT
	VAR_INPUT
		aElement	:	REFERENCE TO TcVnPoint3_LREAL;	(* Element to set at the specified container position *)
		ipContainer	:	ITcVnContainer;	(* Container with TcVnPoint3_LREAL elements, in which the element at position nIndex is replaced by aElement *)
		nIndex	:	ULINT;	(* Index *)
		hrPrev	:	HRESULT;	(* HRESULT indicating the result of previous operations (If SUCCEEDED(hrPrev) equals false, no operation is executed.) *)
	END_VAR

END_FUNCTION

// Functions/Basic Container Operations/F_VN_SetAt/F_VN_SetAt_TcVnPoint3_REAL

	{attribute 'TcIecLibraryType'}
	{attribute 'external_name' := 'F_VN_SetAt_TcVnPoint3_REAL_GUID_E66ACA5D_D15D_444B_607E_3FE1F8E2E557'}
	(* Sets the element at the specified index of the container. *)
	FUNCTION F_VN_SetAt_TcVnPoint3_REAL : HRESULT
	VAR_INPUT
		aElement	:	REFERENCE TO TcVnPoint3_REAL;	(* Element to set at the specified container position *)
		ipContainer	:	ITcVnContainer;	(* Container with TcVnPoint3_REAL elements, in which the element at position nIndex is replaced by aElement *)
		nIndex	:	ULINT;	(* Index *)
		hrPrev	:	HRESULT;	(* HRESULT indicating the result of previous operations (If SUCCEEDED(hrPrev) equals false, no operation is executed.) *)
	END_VAR

END_FUNCTION

// Functions/Basic Container Operations/F_VN_SetAt/F_VN_SetAt_TcVnRectangle_DINT

	{attribute 'TcIecLibraryType'}
	{attribute 'external_name' := 'F_VN_SetAt_TcVnRectangle_DINT_GUID_6A4B7B81_52CE_400A_401D_12D4D52DEFB6'}
	(* Sets the element at the specified index of the container. *)
	FUNCTION F_VN_SetAt_TcVnRectangle_DINT : HRESULT
	VAR_INPUT
		stElement	:	REFERENCE TO TcVnRectangle_DINT;	(* Element to set at the specified container position *)
		ipContainer	:	ITcVnContainer;	(* Container with TcVnRectangle_DINT elements, in which the element at position nIndex is replaced by stElement *)
		nIndex	:	ULINT;	(* Index *)
		hrPrev	:	HRESULT;	(* HRESULT indicating the result of previous operations (If SUCCEEDED(hrPrev) equals false, no operation is executed.) *)
	END_VAR

END_FUNCTION

// Functions/Basic Container Operations/F_VN_SetAt/F_VN_SetAt_TcVnVector2_DINT

	{attribute 'TcIecLibraryType'}
	{attribute 'external_name' := 'F_VN_SetAt_TcVnVector2_DINT_GUID_01E59ECD_1ACB_4A2E_7FC7_8876B067E181'}
	(* Sets the element at the specified index of the container. *)
	FUNCTION F_VN_SetAt_TcVnVector2_DINT : HRESULT
	VAR_INPUT
		aElement	:	REFERENCE TO TcVnVector2_DINT;	(* Element to set at the specified container position *)
		ipContainer	:	ITcVnContainer;	(* Container with TcVnVector2_DINT elements, in which the element at position nIndex is replaced by aElement *)
		nIndex	:	ULINT;	(* Index *)
		hrPrev	:	HRESULT;	(* HRESULT indicating the result of previous operations (If SUCCEEDED(hrPrev) equals false, no operation is executed.) *)
	END_VAR

END_FUNCTION

// Functions/Basic Container Operations/F_VN_SetAt/F_VN_SetAt_TcVnVector2_REAL

	{attribute 'TcIecLibraryType'}
	{attribute 'external_name' := 'F_VN_SetAt_TcVnVector2_REAL_GUID_D3972AA1_11EC_4C98_7BED_57FBEFC33EE6'}
	(* Sets the element at the specified index of the container. *)
	FUNCTION F_VN_SetAt_TcVnVector2_REAL : HRESULT
	VAR_INPUT
		aElement	:	REFERENCE TO TcVnVector2_REAL;	(* Element to set at the specified container position *)
		ipContainer	:	ITcVnContainer;	(* Container with TcVnVector2_REAL elements, in which the element at position nIndex is replaced by aElement *)
		nIndex	:	ULINT;	(* Index *)
		hrPrev	:	HRESULT;	(* HRESULT indicating the result of previous operations (If SUCCEEDED(hrPrev) equals false, no operation is executed.) *)
	END_VAR

END_FUNCTION

// Functions/Basic Container Operations/F_VN_SetAt/F_VN_SetAt_TcVnVector3_REAL

	{attribute 'TcIecLibraryType'}
	{attribute 'external_name' := 'F_VN_SetAt_TcVnVector3_REAL_GUID_C898DEB5_036E_4899_7BEC_82E42720FF9D'}
	(* Sets the element at the specified index of the container. *)
	FUNCTION F_VN_SetAt_TcVnVector3_REAL : HRESULT
	VAR_INPUT
		aElement	:	REFERENCE TO TcVnVector3_REAL;	(* Element to set at the specified container position *)
		ipContainer	:	ITcVnContainer;	(* Container with TcVnVector3_REAL elements, in which the element at position nIndex is replaced by aElement *)
		nIndex	:	ULINT;	(* Index *)
		hrPrev	:	HRESULT;	(* HRESULT indicating the result of previous operations (If SUCCEEDED(hrPrev) equals false, no operation is executed.) *)
	END_VAR

END_FUNCTION

// Functions/Basic Container Operations/F_VN_SetAt/F_VN_SetAt_TcVnVector4_DINT

	{attribute 'TcIecLibraryType'}
	{attribute 'external_name' := 'F_VN_SetAt_TcVnVector4_DINT_GUID_DBE06ADD_9E91_4C53_64A9_E748AFCEFFAC'}
	(* Sets the element at the specified index of the container. *)
	FUNCTION F_VN_SetAt_TcVnVector4_DINT : HRESULT
	VAR_INPUT
		aElement	:	REFERENCE TO TcVnVector4_DINT;	(* Element to set at the specified container position *)
		ipContainer	:	ITcVnContainer;	(* Container with TcVnVector4_DINT elements, in which the element at position nIndex is replaced by aElement *)
		nIndex	:	ULINT;	(* Index *)
		hrPrev	:	HRESULT;	(* HRESULT indicating the result of previous operations (If SUCCEEDED(hrPrev) equals false, no operation is executed.) *)
	END_VAR

END_FUNCTION

// Functions/Basic Container Operations/F_VN_SetAt/F_VN_SetAt_UDINT

	{attribute 'TcIecLibraryType'}
	{attribute 'external_name' := 'F_VN_SetAt_UDINT_GUID_9C7C7581_9250_4E3E_62FC_A17067D710BE'}
	(* Sets the element at the specified index of the container. *)
	FUNCTION F_VN_SetAt_UDINT : HRESULT
	VAR_INPUT
		nElement	:	UDINT;	(* Element to set at the specified container position *)
		ipContainer	:	ITcVnContainer;	(* Container with UDINT elements, in which the element at position nIndex is replaced by nElement *)
		nIndex	:	ULINT;	(* Index *)
		hrPrev	:	HRESULT;	(* HRESULT indicating the result of previous operations (If SUCCEEDED(hrPrev) equals false, no operation is executed.) *)
	END_VAR

END_FUNCTION

// Functions/Basic Container Operations/F_VN_SetAt/F_VN_SetAt_ULINT

	{attribute 'TcIecLibraryType'}
	{attribute 'external_name' := 'F_VN_SetAt_ULINT_GUID_A36F21F2_828A_4D48_5F5F_BE4D49257C30'}
	(* Sets the element at the specified index of the container. *)
	FUNCTION F_VN_SetAt_ULINT : HRESULT
	VAR_INPUT
		nElement	:	ULINT;	(* Element to set at the specified container position *)
		ipContainer	:	ITcVnContainer;	(* Container with ULINT elements, in which the element at position nIndex is replaced by nElement *)
		nIndex	:	ULINT;	(* Index *)
		hrPrev	:	HRESULT;	(* HRESULT indicating the result of previous operations (If SUCCEEDED(hrPrev) equals false, no operation is executed.) *)
	END_VAR

END_FUNCTION

// Functions/Geometric and Coordinate Transformations/Calibration/F_VN_CalibrateCamera

	{attribute 'TcIecLibraryType'}
	{attribute 'external_name' := 'F_VN_CalibrateCamera_GUID_B45668D1_3AE0_4159_4F4F_C62EC011EB27'}
	(* Compute the camera parameters (intrinsic + extrinsic) by evaluating an image containing a calibration pattern (circles). *)
	FUNCTION F_VN_CalibrateCamera : HRESULT
	VAR_INPUT
		ipSrcImage	:	ITcVnImage;	(* Source image containing a calibration pattern (1 channel, USINT elements) *)
		ipReferencePoints	:	ITcVnContainer;	(* Reference calibration pattern point positions (ContainerType_Vector_TcVnPoint3_REAL) *)
		aCameraMatrix	:	REFERENCE TO TcVnMatrix3x3_LREAL;	(* Returns the camera matrix *)
		aDistortionCoefficients	:	REFERENCE TO TcVnArray8_LREAL;	(* Returns the lens distortion coefficients [k1, k2, p1, p2, k3, k4, k5, k6] *)
		aRotationMatrix	:	REFERENCE TO TcVnMatrix3x3_LREAL;	(* Returns the rotation matrix *)
		aTranslationVector	:	REFERENCE TO TcVnVector3_LREAL;	(* Returns the translation vector *)
		fReprojError	:	REFERENCE TO LREAL;	(* Returns the reprojection error *)
		stBlobDetectionParams	:	REFERENCE TO TcVnParamsBlobDetection;	(* Parameters for the internally used F_VN_DetectBlobs function *)
		stCalibrationOptions	:	REFERENCE TO TcVnCameraCalibrationOptions;	(* Calibration options *)
		hrPrev	:	HRESULT;	(* HRESULT indicating the result of previous operations (If SUCCEEDED(hrPrev) equals false, no operation is executed.) *)
	END_VAR

END_FUNCTION

// Functions/Geometric and Coordinate Transformations/Calibration/F_VN_CalibrateCameraExp

	{attribute 'TcIecLibraryType'}
	{attribute 'external_name' := 'F_VN_CalibrateCameraExp_GUID_4283A838_CD7B_4E03_5497_E2B11F84B001'}
	(* Compute the camera parameters (intrinsic + extrinsic) by evaluating images containing a calibration pattern (circles). The extrinsic parameters are computed for the first image in the array. (expert function) *)
	FUNCTION F_VN_CalibrateCameraExp : HRESULT
	VAR_INPUT
		pSrcImages	:	PVOID;	(* Pointer to an array of source images, each containing the same calibration pattern (1 channel, USINT elements) *)
		nSrcArraySize	:	UINT;	(* pSrcImages array size *)
		ipReferencePoints	:	ITcVnContainer;	(* Reference calibration pattern point positions (ContainerType_Vector_TcVnPoint3_REAL) *)
		aCameraMatrix	:	REFERENCE TO TcVnMatrix3x3_LREAL;	(* Returns the camera matrix *)
		aDistortionCoefficients	:	REFERENCE TO TcVnArray8_LREAL;	(* Returns the lens distortion coefficients [k1, k2, p1, p2, k3, k4, k5, k6] *)
		aRotationMatrix	:	REFERENCE TO TcVnMatrix3x3_LREAL;	(* Returns the rotation matrix *)
		aTranslationVector	:	REFERENCE TO TcVnVector3_LREAL;	(* Returns the translation vector *)
		fReprojError	:	REFERENCE TO LREAL;	(* Returns the reprojection error *)
		stBlobDetectionParams	:	REFERENCE TO TcVnParamsBlobDetection;	(* Parameters for the internally used F_VN_DetectBlobs function *)
		stCalibrationOptions	:	REFERENCE TO TcVnCameraCalibrationOptions;	(* Calibration options *)
		hrPrev	:	HRESULT;	(* HRESULT indicating the result of previous operations (If SUCCEEDED(hrPrev) equals false, no operation is executed.) *)
	END_VAR

END_FUNCTION

// Functions/Geometric and Coordinate Transformations/Calibration/F_VN_CalibrateCameraPlanar

